Yaskawa INFORM job: LETTERTR.JBI

/JOB
//NAME LETTERTR
//POS
///NPOS 1576,0,0,0,0,0
///TOOL 0
///POSTYPE PULSE
///PULSE
C00000=-2822,58859,-1118,-1041,-34109,-89
C00001=-2663,58398,-451,-1069,-33796,-147
C00002=-2663,58398,-1851,-1069,-33796,-147
C00003=-2764,58391,-1864,-1056,-33791,-106
C00004=-2845,58329,-1958,-1047,-33753,-73
C00005=-2896,58243,-2089,-1041,-33701,-51
C00006=-2915,58143,-2240,-1040,-33641,-43
C00007=-2900,58040,-2395,-1044,-33578,-47
C00008=-2849,57950,-2529,-1052,-33524,-67
C00009=-2767,57884,-2628,-1064,-33484,-99
C00010=-2668,57851,-2677,-1077,-33464,-138
C00011=-2645,57775,-2791,-1081,-33418,-147
C00012=-2722,57704,-2899,-1072,-33375,-115
C00013=-2807,57646,-2987,-1062,-33340,-80
C00014=-2852,57583,-3083,-1057,-33302,-61
C00015=-2760,57536,-3153,-1070,-33273,-98
C00016=-2666,57492,-3219,-1083,-33246,-135
C00017=-2684,57440,-3296,-1081,-33215,-127
C00018=-2776,57397,-3362,-1070,-33190,-90
C00019=-2811,57371,-3402,-1065,-33174,-75
C00020=-2719,57413,-3338,-1077,-33199,-113
C00021=-2626,57455,-3274,-1089,-33224,-150
C00022=-2618,57352,-3429,-1091,-33162,-152
C00023=-2640,57254,-3577,-1090,-33102,-142
C00024=-2673,57160,-3720,-1087,-33045,-128
C00025=-2712,57067,-3860,-1083,-32989,-111
C00026=-2749,56974,-4000,-1080,-32933,-95
C00027=-2729,56988,-3980,-1082,-32941,-103
C00028=-2696,57083,-3836,-1085,-32999,-118
C00029=-2658,57176,-3696,-1089,-33055,-134
C00030=-2620,57268,-3556,-1092,-33111,-150
C00031=-2574,57251,-3581,-1099,-33100,-168
C00032=-2533,57158,-3722,-1106,-33043,-184
C00033=-2487,57065,-3861,-1113,-32987,-201
C00034=-2437,56975,-3997,-1121,-32931,-220
C00035=-2389,56892,-4124,-1129,-32880,-238
C00036=-2428,56983,-3985,-1122,-32936,-224
C00037=-2479,57073,-3849,-1114,-32991,-205
C00038=-2523,57166,-3710,-1107,-33048,-188
C00039=-2565,57259,-3569,-1100,-33105,-172
C00040=-2606,57348,-3435,-1093,-33159,-157
C00041=-2610,57453,-3277,-1091,-33222,-157
C00042=-2508,57437,-3300,-1105,-33213,-197
C00043=-2406,57411,-3339,-1119,-33196,-238
C00044=-2346,57409,-3342,-1127,-33195,-262
C00045=-2448,57433,-3305,-1113,-33210,-221
C00046=-2551,57457,-3270,-1099,-33225,-180
C00047=-2555,57511,-3189,-1097,-33257,-179
C00048=-2468,57564,-3107,-1108,-33290,-215
C00049=-2400,57631,-3005,-1116,-33330,-243
C00050=-2485,57694,-2912,-1104,-33369,-210
C00051=-2569,57757,-2817,-1092,-33407,-177
C00052=-2616,57836,-2698,-1084,-33455,-159
C00053=-2509,57839,-2693,-1098,-33457,-202
C00054=-2413,57872,-2641,-1111,-33477,-241
C00055=-2340,57940,-2537,-1119,-33519,-271
C00056=-2296,58030,-2401,-1124,-33573,-290
C00057=-2288,58130,-2250,-1123,-33634,-294
C00058=-2316,58227,-2102,-1118,-33694,-284
C00059=-2376,58313,-1975,-1109,-33745,-261
C00060=-2460,58376,-1880,-1097,-33784,-228
C00061=-2561,58402,-1842,-1083,-33799,-188
C00062=-2663,58398,-1851,-1069,-33796,-147
C00063=-2663,58398,-451,-1069,-33796,-147
C00064=-2673,58389,-465,-1068,-33790,-142
C00065=-2673,58389,-1865,-1068,-33790,-142
C00066=-2704,58383,-1875,-1064,-33786,-130
C00067=-2673,58381,-1877,-1068,-33785,-143
C00068=-2641,58379,-1880,-1073,-33784,-155
C00069=-2631,58387,-1866,-1074,-33790,-159
C00070=-2599,58391,-1860,-1078,-33792,-172
C00071=-2566,58392,-1859,-1082,-33793,-186
C00072=-2534,58387,-1865,-1087,-33790,-199
C00073=-2502,58380,-1875,-1091,-33786,-211
C00074=-2471,58371,-1889,-1095,-33780,-224
C00075=-2441,58357,-1909,-1099,-33772,-235
C00076=-2416,58336,-1941,-1103,-33759,-245
C00077=-2392,58314,-1973,-1107,-33746,-255
C00078=-2369,58290,-2009,-1110,-33731,-264
C00079=-2346,58266,-2045,-1113,-33717,-272
C00080=-2331,58237,-2088,-1116,-33700,-278
C00081=-2318,58208,-2131,-1118,-33682,-283
C00082=-2306,58179,-2176,-1120,-33664,-288
C00083=-2301,58147,-2224,-1121,-33645,-289
C00084=-2296,58115,-2272,-1122,-33625,-291
C00085=-2294,58082,-2322,-1123,-33605,-291
C00086=-2300,58051,-2369,-1123,-33586,-288
C00087=-2309,58021,-2415,-1122,-33568,-284
C00088=-2321,57993,-2458,-1121,-33551,-279
C00089=-2336,57966,-2499,-1119,-33534,-273
C00090=-2354,57940,-2538,-1117,-33518,-265
C00091=-2372,57914,-2578,-1115,-33503,-258
C00092=-2398,57894,-2607,-1112,-33491,-247
C00093=-2425,57878,-2632,-1109,-33481,-236
C00094=-2453,57864,-2654,-1105,-33472,-224
C00095=-2483,57854,-2669,-1102,-33466,-212
C00096=-2514,57849,-2678,-1098,-33463,-200
C00097=-2548,57848,-2679,-1093,-33462,-186
C00098=-2581,57848,-2680,-1089,-33462,-173
C00099=-2615,57849,-2679,-1084,-33463,-160
C00100=-2646,57857,-2667,-1080,-33468,-147
C00101=-2678,57864,-2657,-1076,-33472,-134
C00102=-2710,57873,-2644,-1071,-33478,-122
C00103=-2739,57885,-2626,-1067,-33485,-110
C00104=-2769,57898,-2606,-1063,-33493,-98
C00105=-2797,57915,-2582,-1059,-33503,-87
C00106=-2821,57936,-2550,-1056,-33516,-78
C00107=-2843,57961,-2512,-1052,-33531,-69
C00108=-2863,57988,-2473,-1049,-33547,-62
C00109=-2877,58017,-2430,-1047,-33564,-56
C00110=-2889,58046,-2385,-1045,-33582,-52
C00111=-2896,58077,-2338,-1044,-33601,-49
C00112=-2900,58110,-2290,-1043,-33621,-48
C00113=-2903,58143,-2240,-1042,-33640,-47
C00114=-2901,58175,-2191,-1041,-33660,-48
C00115=-2893,58206,-2145,-1042,-33679,-52
C00116=-2885,58236,-2099,-1043,-33697,-56
C00117=-2876,58266,-2053,-1043,-33715,-60
C00118=-2860,58293,-2012,-1045,-33732,-66
C00119=-2840,58318,-1974,-1047,-33747,-75
C00120=-2819,58342,-1938,-1050,-33762,-84
C00121=-2793,58361,-1909,-1053,-33773,-94
C00122=-2766,58377,-1884,-1056,-33783,-105
C00123=-2736,58389,-1866,-1060,-33790,-117
C00124=-2705,58393,-1859,-1064,-33793,-130
C00125=-2673,58389,-1865,-1068,-33790,-142
C00126=-2673,58389,-465,-1068,-33790,-142
C00127=-2757,58271,-644,-1059,-33719,-108
C00128=-2757,58271,-2044,-1059,-33719,-108
C00129=-2762,58267,-2051,-1059,-33716,-106
C00130=-2765,58261,-2060,-1058,-33712,-104
C00131=-2768,58254,-2069,-1058,-33709,-103
C00132=-2769,58248,-2080,-1058,-33704,-102
C00133=-2772,58241,-2089,-1058,-33701,-101
C00134=-2773,58234,-2100,-1057,-33696,-101
C00135=-2775,58228,-2110,-1057,-33692,-100
C00136=-2776,58221,-2120,-1057,-33688,-99
C00137=-2778,58214,-2131,-1057,-33684,-98
C00138=-2779,58207,-2141,-1057,-33680,-98
C00139=-2780,58200,-2152,-1057,-33676,-97
C00140=-2781,58193,-2163,-1057,-33671,-97
C00141=-2781,58185,-2174,-1057,-33667,-97
C00142=-2782,58178,-2185,-1057,-33662,-96
C00143=-2782,58171,-2196,-1057,-33658,-96
C00144=-2783,58164,-2206,-1057,-33654,-96
C00145=-2782,58157,-2217,-1057,-33649,-96
C00146=-2781,58150,-2227,-1058,-33645,-97
C00147=-2780,58143,-2238,-1058,-33641,-97
C00148=-2778,58136,-2248,-1058,-33637,-97
C00149=-2776,58129,-2259,-1059,-33633,-98
C00150=-2774,58123,-2268,-1059,-33629,-99
C00151=-2770,58116,-2278,-1060,-33625,-100
C00152=-2767,58110,-2287,-1060,-33621,-102
C00153=-2762,58104,-2296,-1061,-33618,-103
C00154=-2757,58100,-2302,-1062,-33615,-106
C00155=-2750,58097,-2307,-1063,-33613,-108
C00156=-2744,58095,-2310,-1063,-33612,-111
C00157=-2738,58091,-2315,-1064,-33610,-113
C00158=-2731,58090,-2317,-1065,-33609,-116
C00159=-2724,58092,-2314,-1066,-33610,-119
C00160=-2718,58096,-2308,-1067,-33612,-121
C00161=-2713,58100,-2301,-1067,-33615,-123
C00162=-2711,58107,-2291,-1068,-33619,-124
C00163=-2710,58114,-2281,-1068,-33623,-124
C00164=-2708,58120,-2271,-1068,-33627,-125
C00165=-2704,58126,-2262,-1068,-33631,-127
C00166=-2704,58134,-2251,-1068,-33635,-127
C00167=-2704,58141,-2240,-1068,-33640,-127
C00168=-2705,58148,-2229,-1068,-33644,-127
C00169=-2706,58155,-2219,-1067,-33648,-126
C00170=-2707,58162,-2208,-1067,-33653,-126
C00171=-2707,58169,-2198,-1067,-33657,-126
C00172=-2710,58175,-2188,-1067,-33661,-125
C00173=-2710,58183,-2177,-1067,-33665,-126
C00174=-2712,58189,-2167,-1066,-33669,-125
C00175=-2713,58196,-2157,-1066,-33673,-124
C00176=-2716,58202,-2147,-1065,-33677,-123
C00177=-2718,58209,-2137,-1065,-33681,-122
C00178=-2720,58216,-2127,-1065,-33685,-122
C00179=-2722,58222,-2117,-1064,-33689,-121
C00180=-2724,58229,-2107,-1064,-33693,-120
C00181=-2727,58236,-2097,-1064,-33697,-119
C00182=-2733,58239,-2092,-1063,-33699,-117
C00183=-2738,58244,-2084,-1062,-33703,-115
C00184=-2740,58251,-2074,-1062,-33706,-114
C00185=-2743,58257,-2064,-1061,-33710,-113
C00186=-2745,58264,-2054,-1061,-33715,-112
C00187=-2750,58269,-2048,-1060,-33717,-110
C00188=-2757,58271,-2044,-1059,-33719,-108
C00189=-2757,58271,-644,-1059,-33719,-108
C00190=-2516,58232,-699,-1091,-33696,-204
C00191=-2516,58232,-2099,-1091,-33696,-204
C00192=-2518,58225,-2110,-1091,-33691,-203
C00193=-2519,58217,-2121,-1091,-33687,-203
C00194=-2521,58210,-2132,-1091,-33683,-202
C00195=-2522,58203,-2143,-1091,-33678,-201
C00196=-2523,58196,-2154,-1091,-33674,-201
C00197=-2525,58189,-2164,-1091,-33669,-200
C00198=-2526,58181,-2176,-1091,-33665,-199
C00199=-2527,58174,-2187,-1091,-33661,-199
C00200=-2527,58166,-2199,-1091,-33656,-198
C00201=-2527,58158,-2210,-1091,-33651,-198
C00202=-2528,58151,-2222,-1091,-33646,-198
C00203=-2526,58143,-2233,-1091,-33642,-199
C00204=-2525,58136,-2244,-1092,-33637,-199
C00205=-2522,58129,-2254,-1092,-33633,-200
C00206=-2518,58123,-2264,-1093,-33629,-201
C00207=-2516,58116,-2274,-1093,-33625,-202
C00208=-2513,58109,-2285,-1094,-33621,-203
C00209=-2511,58102,-2295,-1094,-33617,-204
C00210=-2507,58096,-2305,-1095,-33613,-206
C00211=-2504,58089,-2314,-1095,-33609,-207
C00212=-2500,58083,-2324,-1096,-33605,-208
C00213=-2495,58077,-2333,-1097,-33601,-210
C00214=-2490,58071,-2342,-1097,-33598,-212
C00215=-2484,58066,-2349,-1098,-33595,-214
C00216=-2478,58063,-2354,-1099,-33593,-217
C00217=-2470,58063,-2354,-1100,-33593,-220
C00218=-2465,58068,-2345,-1101,-33596,-222
C00219=-2462,58074,-2336,-1101,-33600,-224
C00220=-2458,58081,-2327,-1101,-33604,-225
C00221=-2455,58087,-2317,-1102,-33608,-226
C00222=-2453,58094,-2307,-1102,-33612,-228
C00223=-2452,58101,-2295,-1102,-33617,-228
C00224=-2451,58109,-2284,-1102,-33621,-229
C00225=-2450,58116,-2272,-1102,-33626,-229
C00226=-2450,58124,-2261,-1102,-33631,-229
C00227=-2451,58132,-2249,-1102,-33635,-229
C00228=-2451,58140,-2238,-1101,-33640,-229
C00229=-2451,58147,-2226,-1101,-33645,-229
C00230=-2452,58154,-2215,-1101,-33649,-228
C00231=-2453,58162,-2204,-1101,-33653,-228
C00232=-2455,58169,-2193,-1100,-33658,-228
C00233=-2457,58176,-2182,-1100,-33662,-227
C00234=-2458,58183,-2171,-1100,-33666,-226
C00235=-2460,58191,-2160,-1099,-33671,-226
C00236=-2462,58198,-2150,-1099,-33675,-225
C00237=-2464,58205,-2140,-1099,-33679,-224
C00238=-2466,58212,-2129,-1098,-33684,-224
C00239=-2468,58219,-2118,-1098,-33688,-223
C00240=-2470,58226,-2107,-1098,-33692,-222
C00241=-2474,58232,-2098,-1097,-33696,-221
C00242=-2477,58239,-2088,-1096,-33700,-220
C00243=-2479,58246,-2078,-1096,-33704,-219
C00244=-2482,58253,-2067,-1096,-33708,-218
C00245=-2486,58258,-2059,-1095,-33712,-216
C00246=-2494,58260,-2057,-1094,-33713,-213
C00247=-2500,58256,-2063,-1093,-33710,-211
C00248=-2504,58250,-2072,-1093,-33707,-209
C00249=-2508,58244,-2081,-1092,-33703,-207
C00250=-2513,58238,-2090,-1092,-33700,-205
C00251=-2516,58232,-2099,-1091,-33696,-204
C00252=-2516,58232,-699,-1091,-33696,-204
C00253=-2186,58255,-658,-1135,-33711,-337
C00254=-2186,58255,-2058,-1135,-33711,-337
C00255=-2183,58242,-2078,-1135,-33703,-338
C00256=-2179,58229,-2098,-1136,-33695,-339
C00257=-2171,58217,-2115,-1137,-33688,-342
C00258=-2162,58207,-2131,-1138,-33682,-346
C00259=-2150,58199,-2143,-1140,-33677,-350
C00260=-2137,58196,-2148,-1142,-33675,-356
C00261=-2124,58198,-2143,-1144,-33677,-361
C00262=-2112,58204,-2134,-1145,-33680,-366
C00263=-2103,58215,-2118,-1146,-33687,-369
C00264=-2097,58227,-2100,-1147,-33694,-372
C00265=-2098,58239,-2081,-1146,-33701,-372
C00266=-2106,58247,-2069,-1145,-33707,-369
C00267=-2108,58234,-2089,-1145,-33698,-368
C00268=-2111,58221,-2109,-1145,-33690,-366
C00269=-2121,58211,-2124,-1144,-33684,-362
C00270=-2133,58205,-2133,-1142,-33681,-357
C00271=-2147,58206,-2132,-1140,-33681,-352
C00272=-2158,58215,-2118,-1139,-33687,-347
C00273=-2167,58226,-2101,-1138,-33694,-344
C00274=-2173,58239,-2083,-1137,-33701,-342
C00275=-2176,58252,-2063,-1136,-33709,-341
C00276=-2179,58265,-2043,-1135,-33717,-340
C00277=-2181,58279,-2022,-1135,-33726,-339
C00278=-2182,58293,-2001,-1134,-33734,-339
C00279=-2183,58307,-1979,-1134,-33743,-339
C00280=-2181,58321,-1959,-1134,-33751,-340
C00281=-2178,58334,-1939,-1134,-33759,-341
C00282=-2173,58346,-1920,-1135,-33767,-343
C00283=-2168,58359,-1901,-1135,-33774,-345
C00284=-2160,58369,-1885,-1136,-33781,-349
C00285=-2151,58380,-1869,-1137,-33787,-353
C00286=-2138,58385,-1861,-1139,-33791,-358
C00287=-2124,58384,-1862,-1141,-33790,-363
C00288=-2111,58381,-1867,-1142,-33788,-368
C00289=-2104,58370,-1883,-1143,-33782,-371
C00290=-2099,58357,-1902,-1144,-33774,-373
C00291=-2096,58344,-1922,-1145,-33766,-374
C00292=-2093,58330,-1943,-1145,-33757,-375
C00293=-2092,58317,-1964,-1146,-33749,-375
C00294=-2081,58320,-1959,-1147,-33751,-380
C00295=-2082,58333,-1939,-1147,-33759,-379
C00296=-2085,58346,-1919,-1146,-33767,-379
C00297=-2089,58359,-1899,-1146,-33775,-377
C00298=-2093,58372,-1879,-1145,-33783,-376
C00299=-2097,58385,-1860,-1144,-33791,-374
C00300=-2108,58391,-1850,-1143,-33795,-370
C00301=-2122,58395,-1845,-1141,-33797,-364
C00302=-2137,58396,-1844,-1139,-33797,-358
C00303=-2150,58393,-1849,-1137,-33795,-353
C00304=-2161,58385,-1862,-1136,-33790,-348
C00305=-2170,58374,-1878,-1135,-33784,-345
C00306=-2175,58362,-1896,-1134,-33776,-342
C00307=-2182,58351,-1914,-1134,-33769,-340
C00308=-2186,58338,-1933,-1133,-33762,-338
C00309=-2189,58325,-1953,-1133,-33754,-336
C00310=-2191,58311,-1974,-1133,-33745,-335
C00311=-2190,58297,-1995,-1133,-33737,-335
C00312=-2190,58283,-2016,-1134,-33728,-336
C00313=-2188,58269,-2037,-1134,-33720,-336
C00314=-2186,58255,-2058,-1135,-33711,-337
C00315=-2186,58255,-658,-1135,-33711,-337
C00316=-2073,58248,-667,-1150,-33707,-382
C00317=-2073,58248,-2067,-1150,-33707,-382
C00318=-2072,58241,-2077,-1150,-33703,-382
C00319=-2071,58235,-2087,-1150,-33699,-383
C00320=-2069,58229,-2096,-1150,-33695,-383
C00321=-2067,58223,-2105,-1151,-33692,-384
C00322=-2063,58217,-2114,-1151,-33688,-385
C00323=-2059,58212,-2121,-1152,-33685,-387
C00324=-2053,58209,-2126,-1153,-33683,-390
C00325=-2047,58206,-2130,-1154,-33682,-392
C00326=-2041,58203,-2135,-1154,-33680,-394
C00327=-2035,58202,-2137,-1155,-33679,-397
C00328=-2028,58202,-2136,-1156,-33679,-399
C00329=-2021,58202,-2136,-1157,-33679,-402
C00330=-2015,58205,-2131,-1158,-33681,-405
C00331=-2010,58209,-2125,-1158,-33683,-407
C00332=-2006,58214,-2118,-1159,-33687,-409
C00333=-2003,58219,-2109,-1159,-33690,-410
C00334=-2001,58225,-2100,-1159,-33694,-411
C00335=-1999,58231,-2091,-1160,-33697,-412
C00336=-1999,58238,-2080,-1159,-33702,-412
C00337=-1994,58236,-2083,-1160,-33701,-413
C00338=-1993,58230,-2093,-1160,-33697,-414
C00339=-1990,58224,-2101,-1161,-33693,-415
C00340=-1987,58218,-2110,-1161,-33689,-416
C00341=-1985,58212,-2120,-1162,-33686,-417
C00342=-1984,58206,-2129,-1162,-33682,-417
C00343=-1981,58200,-2139,-1162,-33678,-418
C00344=-1976,58196,-2144,-1163,-33676,-420
C00345=-1969,58198,-2142,-1164,-33677,-423
C00346=-1969,58204,-2132,-1164,-33681,-423
C00347=-1973,58209,-2124,-1163,-33684,-422
C00348=-1976,58215,-2115,-1163,-33687,-421
C00349=-1978,58221,-2106,-1162,-33691,-420
C00350=-1980,58227,-2097,-1162,-33695,-419
C00351=-1982,58233,-2088,-1162,-33699,-418
C00352=-1985,58239,-2079,-1161,-33702,-417
C00353=-1987,58245,-2069,-1161,-33706,-417
C00354=-1989,58251,-2060,-1160,-33710,-416
C00355=-1990,58258,-2050,-1160,-33714,-415
C00356=-1992,58264,-2041,-1160,-33718,-415
C00357=-1994,58270,-2032,-1160,-33721,-414
C00358=-1995,58277,-2022,-1159,-33725,-414
C00359=-1998,58283,-2013,-1159,-33729,-413
C00360=-2001,58289,-2004,-1158,-33732,-412
C00361=-2006,58290,-2002,-1158,-33733,-409
C00362=-2012,58292,-2000,-1157,-33734,-407
C00363=-2017,58297,-1992,-1156,-33737,-405
C00364=-2022,58302,-1985,-1155,-33740,-403
C00365=-2029,58303,-1983,-1154,-33741,-401
C00366=-2036,58304,-1982,-1154,-33741,-398
C00367=-2042,58302,-1985,-1153,-33740,-395
C00368=-2047,58298,-1990,-1152,-33738,-393
C00369=-2052,58294,-1997,-1152,-33735,-391
C00370=-2057,58289,-2004,-1151,-33733,-389
C00371=-2061,58284,-2012,-1151,-33729,-387
C00372=-2064,58279,-2020,-1150,-33726,-386
C00373=-2067,58273,-2029,-1150,-33723,-385
C00374=-2069,58267,-2038,-1150,-33719,-384
C00375=-2071,58261,-2047,-1150,-33715,-383
C00376=-2072,58255,-2057,-1150,-33711,-383
C00377=-2073,58248,-2067,-1150,-33707,-382
C00378=-2073,58248,-667,-1150,-33707,-382
C00379=-2064,58248,-666,-1151,-33708,-386
C00380=-2064,58248,-2066,-1151,-33708,-386
C00381=-2063,58252,-2061,-1151,-33710,-386
C00382=-2062,58256,-2055,-1151,-33712,-387
C00383=-2061,58259,-2050,-1151,-33714,-387
C00384=-2060,58263,-2045,-1151,-33716,-388
C00385=-2059,58266,-2039,-1151,-33718,-388
C00386=-2057,58269,-2035,-1151,-33720,-389
C00387=-2056,58273,-2029,-1151,-33722,-389
C00388=-2054,58276,-2024,-1152,-33724,-390
C00389=-2051,58278,-2021,-1152,-33726,-391
C00390=-2050,58281,-2016,-1152,-33728,-392
C00391=-2048,58285,-2011,-1152,-33730,-393
C00392=-2046,58287,-2007,-1152,-33731,-394
C00393=-2042,58289,-2004,-1153,-33733,-395
C00394=-2039,58291,-2001,-1153,-33734,-396
C00395=-2036,58292,-2000,-1154,-33734,-398
C00396=-2032,58293,-1998,-1154,-33735,-399
C00397=-2028,58294,-1997,-1155,-33736,-400
C00398=-2025,58292,-2000,-1155,-33734,-402
C00399=-2022,58289,-2003,-1156,-33733,-403
C00400=-2019,58287,-2007,-1156,-33731,-404
C00401=-2016,58285,-2010,-1156,-33730,-405
C00402=-2013,58282,-2014,-1157,-33729,-407
C00403=-2010,58280,-2017,-1157,-33727,-408
C00404=-2009,58277,-2023,-1158,-33725,-408
C00405=-2008,58273,-2028,-1158,-33723,-409
C00406=-2007,58269,-2033,-1158,-33721,-409
C00407=-2007,58265,-2039,-1158,-33718,-409
C00408=-2006,58262,-2044,-1158,-33716,-409
C00409=-2007,58258,-2050,-1158,-33714,-409
C00410=-2007,58255,-2055,-1158,-33712,-408
C00411=-2007,58251,-2061,-1158,-33709,-409
C00412=-2008,58248,-2067,-1158,-33707,-408
C00413=-2008,58244,-2072,-1158,-33705,-408
C00414=-2008,58240,-2078,-1158,-33702,-408
C00415=-2008,58236,-2084,-1158,-33700,-408
C00416=-2009,58232,-2090,-1158,-33698,-407
C00417=-2010,58229,-2095,-1158,-33696,-407
C00418=-2011,58225,-2101,-1158,-33694,-407
C00419=-2012,58222,-2106,-1158,-33691,-406
C00420=-2015,58219,-2110,-1158,-33690,-405
C00421=-2017,58216,-2115,-1157,-33688,-404
C00422=-2020,58213,-2118,-1157,-33686,-403
C00423=-2023,58211,-2122,-1157,-33685,-402
C00424=-2026,58210,-2124,-1156,-33684,-400
C00425=-2030,58209,-2125,-1156,-33684,-399
C00426=-2034,58210,-2124,-1155,-33684,-397
C00427=-2038,58211,-2123,-1155,-33685,-396
C00428=-2041,58212,-2121,-1154,-33685,-394
C00429=-2045,58213,-2119,-1154,-33686,-393
C00430=-2048,58216,-2116,-1153,-33688,-392
C00431=-2051,58218,-2112,-1153,-33689,-390
C00432=-2054,58220,-2109,-1152,-33690,-389
C00433=-2056,58223,-2104,-1152,-33692,-388
C00434=-2058,58227,-2099,-1152,-33694,-388
C00435=-2060,58230,-2094,-1152,-33696,-387
C00436=-2061,58233,-2089,-1151,-33698,-386
C00437=-2062,58237,-2083,-1151,-33701,-386
C00438=-2062,58241,-2077,-1151,-33703,-386
C00439=-2063,58245,-2072,-1151,-33705,-386
C00440=-2064,58248,-2066,-1151,-33708,-386
C00441=-2064,58248,-666,-1151,-33708,-386
C00442=-1952,58261,-646,-1165,-33715,-431
C00443=-1952,58261,-2046,-1165,-33715,-431
C00444=-1950,58252,-2059,-1166,-33710,-432
C00445=-1948,58243,-2072,-1166,-33705,-432
C00446=-1946,58234,-2086,-1166,-33699,-433
C00447=-1944,58225,-2099,-1167,-33694,-433
C00448=-1943,58216,-2113,-1167,-33688,-434
C00449=-1942,58207,-2127,-1167,-33683,-434
C00450=-1941,58198,-2140,-1168,-33677,-435
C00451=-1936,58190,-2152,-1168,-33672,-436
C00452=-1928,58190,-2152,-1170,-33673,-439
C00453=-1927,58200,-2138,-1169,-33678,-440
C00454=-1929,58208,-2124,-1169,-33684,-439
C00455=-1931,58217,-2111,-1169,-33689,-439
C00456=-1932,58227,-2097,-1169,-33695,-439
C00457=-1932,58236,-2083,-1168,-33700,-438
C00458=-1933,58245,-2069,-1168,-33706,-438
C00459=-1930,58253,-2056,-1168,-33711,-439
C00460=-1927,58262,-2044,-1168,-33716,-441
C00461=-1924,58270,-2032,-1169,-33721,-442
C00462=-1917,58276,-2022,-1170,-33725,-445
C00463=-1908,58279,-2017,-1171,-33727,-449
C00464=-1899,58280,-2015,-1172,-33728,-452
C00465=-1891,58276,-2021,-1173,-33725,-455
C00466=-1884,58270,-2031,-1174,-33721,-458
C00467=-1878,58262,-2042,-1175,-33717,-460
C00468=-1873,58254,-2054,-1176,-33712,-462
C00469=-1870,58246,-2066,-1176,-33707,-464
C00470=-1867,58238,-2079,-1177,-33702,-465
C00471=-1864,58229,-2092,-1177,-33697,-466
C00472=-1862,58220,-2105,-1178,-33691,-466
C00473=-1860,58211,-2119,-1178,-33686,-467
C00474=-1860,58202,-2133,-1178,-33680,-467
C00475=-1856,58194,-2145,-1179,-33675,-468
C00476=-1847,58196,-2142,-1180,-33676,-472
C00477=-1846,58205,-2128,-1180,-33682,-473
C00478=-1848,58214,-2115,-1180,-33687,-472
C00479=-1851,58222,-2102,-1179,-33692,-471
C00480=-1855,58230,-2090,-1179,-33697,-470
C00481=-1857,58239,-2077,-1178,-33703,-469
C00482=-1860,58248,-2064,-1178,-33708,-468
C00483=-1863,58256,-2051,-1177,-33713,-466
C00484=-1867,58264,-2039,-1176,-33718,-465
C00485=-1873,58271,-2028,-1175,-33722,-463
C00486=-1879,58279,-2017,-1175,-33727,-460
C00487=-1886,58285,-2007,-1174,-33731,-458
C00488=-1894,58290,-2000,-1172,-33734,-455
C00489=-1904,58290,-2000,-1171,-33734,-451
C00490=-1912,58288,-2003,-1170,-33733,-447
C00491=-1920,58285,-2008,-1169,-33731,-444
C00492=-1928,58279,-2017,-1168,-33727,-441
C00493=-1933,58272,-2028,-1168,-33723,-439
C00494=-1936,58264,-2040,-1167,-33718,-437
C00495=-1942,58259,-2048,-1167,-33715,-435
C00496=-1945,58268,-2035,-1166,-33720,-434
C00497=-1947,58277,-2022,-1166,-33725,-433
C00498=-1950,58285,-2009,-1165,-33730,-432
C00499=-1955,58292,-1999,-1164,-33734,-430
C00500=-1961,58286,-2007,-1164,-33731,-428
C00501=-1959,58277,-2021,-1164,-33726,-428
C00502=-1956,58269,-2033,-1165,-33721,-429
C00503=-1952,58261,-2046,-1165,-33715,-431
C00504=-1952,58261,-646,-1165,-33715,-431
C00505=-1708,58270,-628,-1197,-33722,-529
C00506=-1708,58270,-2028,-1197,-33722,-529
C00507=-1705,58252,-2054,-1198,-33712,-530
C00508=-1700,58236,-2078,-1199,-33702,-532
C00509=-1693,58220,-2102,-1200,-33692,-534
C00510=-1682,58206,-2123,-1202,-33683,-538
C00511=-1666,58200,-2132,-1204,-33680,-545
C00512=-1651,58208,-2121,-1206,-33684,-551
C00513=-1645,58223,-2098,-1206,-33694,-554
C00514=-1642,58239,-2072,-1206,-33704,-555
C00515=-1645,58257,-2046,-1206,-33714,-554
C00516=-1633,58247,-2061,-1207,-33708,-559
C00517=-1622,58233,-2082,-1209,-33700,-563
C00518=-1612,58218,-2104,-1211,-33691,-567
C00519=-1604,58203,-2127,-1212,-33681,-570
C00520=-1597,58187,-2151,-1213,-33672,-572
C00521=-1595,58170,-2177,-1214,-33661,-573
C00522=-1596,58152,-2204,-1214,-33650,-572
C00523=-1603,58137,-2227,-1213,-33641,-569
C00524=-1611,58123,-2249,-1212,-33632,-566
C00525=-1624,58111,-2268,-1211,-33625,-561
C00526=-1638,58102,-2281,-1209,-33619,-555
C00527=-1655,58105,-2277,-1207,-33621,-548
C00528=-1670,58114,-2263,-1205,-33627,-542
C00529=-1682,58128,-2243,-1203,-33635,-537
C00530=-1694,58142,-2221,-1201,-33644,-533
C00531=-1703,58157,-2199,-1200,-33653,-530
C00532=-1710,58169,-2180,-1199,-33660,-527
C00533=-1705,58153,-2205,-1200,-33650,-529
C00534=-1697,58138,-2228,-1201,-33641,-532
C00535=-1687,58123,-2250,-1203,-33632,-536
C00536=-1675,58110,-2270,-1204,-33624,-540
C00537=-1661,58099,-2286,-1206,-33617,-546
C00538=-1644,58094,-2293,-1209,-33614,-552
C00539=-1627,58097,-2289,-1211,-33616,-559
C00540=-1612,58106,-2275,-1213,-33622,-565
C00541=-1601,58119,-2255,-1214,-33630,-570
C00542=-1592,58133,-2233,-1215,-33639,-574
C00543=-1587,58149,-2209,-1215,-33648,-576
C00544=-1584,58166,-2183,-1215,-33659,-578
C00545=-1586,58183,-2157,-1215,-33669,-577
C00546=-1591,58199,-2133,-1214,-33679,-575
C00547=-1598,58215,-2109,-1213,-33689,-572
C00548=-1607,58230,-2086,-1211,-33698,-569
C00549=-1617,58244,-2065,-1210,-33707,-565
C00550=-1628,58258,-2044,-1208,-33715,-561
C00551=-1640,58272,-2023,-1206,-33724,-556
C00552=-1648,58287,-2000,-1205,-33733,-553
C00553=-1658,58282,-2009,-1204,-33730,-549
C00554=-1654,58265,-2034,-1204,-33720,-551
C00555=-1652,58248,-2060,-1205,-33709,-551
C00556=-1651,58231,-2086,-1205,-33698,-551
C00557=-1656,58215,-2110,-1205,-33689,-549
C00558=-1671,58211,-2116,-1203,-33686,-543
C00559=-1683,58222,-2099,-1201,-33693,-538
C00560=-1690,58238,-2075,-1200,-33703,-536
C00561=-1694,58255,-2050,-1199,-33713,-534
C00562=-1697,58272,-2024,-1199,-33723,-533
C00563=-1697,58290,-1997,-1198,-33735,-534
C00564=-1705,58303,-1978,-1197,-33742,-530
C00565=-1709,58287,-2001,-1197,-33733,-529
C00566=-1708,58270,-2028,-1197,-33722,-529
C00567=-1708,58270,-628,-1197,-33722,-529
C00568=-1590,58245,-662,-1213,-33708,-576
C00569=-1590,58245,-2062,-1213,-33708,-576
C00570=-1592,58236,-2076,-1213,-33702,-575
C00571=-1593,58227,-2090,-1213,-33696,-575
C00572=-1592,58218,-2104,-1213,-33691,-575
C00573=-1588,58209,-2118,-1214,-33685,-576
C00574=-1586,58200,-2131,-1215,-33680,-577
C00575=-1579,58193,-2142,-1215,-33675,-580
C00576=-1574,58185,-2155,-1216,-33670,-582
C00577=-1568,58178,-2165,-1217,-33666,-584
C00578=-1560,58172,-2174,-1218,-33663,-587
C00579=-1551,58168,-2179,-1220,-33661,-591
C00580=-1542,58166,-2182,-1221,-33659,-594
C00581=-1532,58166,-2181,-1222,-33659,-598
C00582=-1523,58169,-2176,-1223,-33661,-602
C00583=-1516,58174,-2169,-1224,-33664,-605
C00584=-1511,58182,-2157,-1225,-33669,-607
C00585=-1509,58191,-2144,-1225,-33675,-608
C00586=-1508,58200,-2129,-1225,-33680,-608
C00587=-1509,58210,-2115,-1224,-33686,-608
C00588=-1511,58219,-2101,-1224,-33692,-608
C00589=-1513,58228,-2087,-1224,-33697,-607
C00590=-1517,58237,-2074,-1223,-33703,-605
C00591=-1520,58245,-2061,-1222,-33708,-604
C00592=-1526,58253,-2049,-1221,-33713,-602
C00593=-1531,58261,-2037,-1221,-33718,-600
C00594=-1538,58268,-2026,-1220,-33722,-597
C00595=-1544,58276,-2015,-1219,-33727,-595
C00596=-1552,58281,-2007,-1218,-33730,-592
C00597=-1550,58272,-2021,-1218,-33724,-592
C00598=-1543,58265,-2032,-1219,-33720,-595
C00599=-1537,58257,-2043,-1220,-33715,-597
C00600=-1532,58249,-2056,-1221,-33710,-599
C00601=-1528,58241,-2068,-1221,-33705,-601
C00602=-1524,58232,-2081,-1222,-33700,-602
C00603=-1521,58224,-2094,-1223,-33695,-604
C00604=-1519,58215,-2108,-1223,-33689,-604
C00605=-1517,58205,-2122,-1223,-33683,-605
C00606=-1518,58196,-2136,-1223,-33678,-604
C00607=-1520,58187,-2150,-1223,-33672,-603
C00608=-1526,58180,-2161,-1223,-33668,-601
C00609=-1534,58177,-2166,-1222,-33666,-597
C00610=-1544,58177,-2165,-1220,-33666,-594
C00611=-1553,58180,-2162,-1219,-33667,-590
C00612=-1561,58185,-2153,-1218,-33671,-587
C00613=-1567,58192,-2143,-1217,-33675,-584
C00614=-1572,58200,-2131,-1216,-33680,-582
C00615=-1577,58208,-2118,-1215,-33685,-581
C00616=-1580,58217,-2105,-1215,-33690,-580
C00617=-1582,58226,-2091,-1215,-33696,-579
C00618=-1581,58236,-2077,-1215,-33702,-580
C00619=-1579,58245,-2063,-1215,-33707,-581
C00620=-1574,58252,-2051,-1215,-33712,-583
C00621=-1567,58259,-2042,-1216,-33716,-586
C00622=-1558,58260,-2040,-1217,-33717,-589
C00623=-1552,58259,-2042,-1218,-33716,-592
C00624=-1556,58267,-2029,-1217,-33721,-590
C00625=-1565,58270,-2025,-1216,-33723,-587
C00626=-1573,58267,-2029,-1215,-33721,-583
C00627=-1581,58261,-2038,-1214,-33718,-580
C00628=-1586,58254,-2050,-1214,-33713,-578
C00629=-1590,58245,-2062,-1213,-33708,-576
C00630=-1590,58245,-662,-1213,-33708,-576
C00631=-1499,58245,-662,-1225,-33708,-613
C00632=-1499,58245,-2062,-1225,-33708,-613
C00633=-1497,58235,-2076,-1226,-33702,-613
C00634=-1495,58226,-2090,-1226,-33696,-614
C00635=-1493,58217,-2104,-1226,-33691,-615
C00636=-1490,58208,-2118,-1227,-33685,-616
C00637=-1487,58199,-2131,-1228,-33680,-617
C00638=-1481,58191,-2143,-1228,-33675,-619
C00639=-1476,58183,-2155,-1229,-33670,-621
C00640=-1468,58176,-2165,-1230,-33666,-624
C00641=-1460,58171,-2174,-1232,-33662,-627
C00642=-1452,58166,-2181,-1233,-33659,-630
C00643=-1444,58161,-2187,-1234,-33657,-634
C00644=-1434,58160,-2189,-1235,-33656,-637
C00645=-1424,58160,-2190,-1236,-33656,-641
C00646=-1415,58162,-2186,-1238,-33657,-645
C00647=-1408,58169,-2176,-1238,-33661,-648
C00648=-1404,58176,-2164,-1239,-33666,-650
C00649=-1401,58185,-2151,-1239,-33671,-651
C00650=-1400,58195,-2136,-1239,-33677,-652
C00651=-1399,58204,-2121,-1239,-33683,-652
C00652=-1399,58214,-2106,-1239,-33689,-653
C00653=-1399,58224,-2092,-1239,-33695,-652
C00654=-1402,58233,-2078,-1238,-33701,-651
C00655=-1404,58242,-2064,-1238,-33707,-651
C00656=-1407,58251,-2050,-1237,-33712,-650
C00657=-1410,58260,-2037,-1237,-33718,-649
C00658=-1413,58269,-2023,-1236,-33723,-648
C00659=-1417,58277,-2010,-1235,-33728,-646
C00660=-1422,58285,-1999,-1235,-33733,-644
C00661=-1429,58291,-1990,-1234,-33737,-641
C00662=-1429,58282,-2004,-1234,-33731,-641
C00663=-1425,58273,-2017,-1234,-33726,-643
C00664=-1421,58265,-2030,-1235,-33720,-644
C00665=-1418,58256,-2043,-1236,-33715,-645
C00666=-1416,58247,-2057,-1236,-33709,-646
C00667=-1413,58238,-2071,-1237,-33704,-647
C00668=-1411,58229,-2085,-1237,-33698,-648
C00669=-1409,58219,-2099,-1237,-33692,-649
C00670=-1409,58210,-2113,-1238,-33687,-648
C00671=-1409,58200,-2128,-1238,-33681,-648
C00672=-1411,58191,-2142,-1238,-33675,-647
C00673=-1413,58182,-2156,-1238,-33669,-646
C00674=-1417,58174,-2168,-1237,-33664,-644
C00675=-1426,58169,-2175,-1236,-33662,-641
C00676=-1435,58169,-2175,-1235,-33661,-637
C00677=-1444,58173,-2170,-1234,-33664,-634
C00678=-1452,58178,-2162,-1232,-33667,-630
C00679=-1460,58184,-2154,-1231,-33670,-627
C00680=-1468,58190,-2144,-1230,-33674,-624
C00681=-1474,58198,-2132,-1229,-33679,-622
C00682=-1478,58207,-2119,-1229,-33684,-620
C00683=-1482,58215,-2106,-1228,-33690,-619
C00684=-1484,58224,-2092,-1227,-33695,-618
C00685=-1486,58234,-2078,-1227,-33701,-618
C00686=-1488,58243,-2064,-1227,-33707,-617
C00687=-1490,58252,-2050,-1226,-33713,-617
C00688=-1489,58262,-2034,-1226,-33719,-617
C00689=-1495,58269,-2025,-1225,-33722,-614
C00690=-1502,58263,-2034,-1224,-33719,-612
C00691=-1500,58254,-2047,-1225,-33714,-612
C00692=-1499,58245,-2062,-1225,-33708,-613
C00693=-1499,58245,-662,-1225,-33708,-613
C00694=-1517,58080,-913,-1226,-33606,-603
C00695=-1517,58080,-2313,-1226,-33606,-603
C00696=-1518,58057,-2347,-1226,-33592,-603
C00697=-1512,58035,-2380,-1227,-33579,-604
C00698=-1507,58014,-2413,-1228,-33565,-606
C00699=-1510,57996,-2440,-1228,-33554,-605
C00700=-1534,57998,-2437,-1225,-33556,-595
C00701=-1541,57990,-2449,-1224,-33551,-592
C00702=-1518,57987,-2454,-1227,-33549,-602
C00703=-1501,57976,-2470,-1230,-33542,-608
C00704=-1497,57954,-2503,-1230,-33529,-609
C00705=-1494,57932,-2538,-1231,-33515,-610
C00706=-1495,57909,-2573,-1232,-33501,-610
C00707=-1483,57902,-2582,-1233,-33497,-614
C00708=-1484,57925,-2548,-1233,-33511,-614
C00709=-1486,57948,-2513,-1232,-33525,-614
C00710=-1490,57970,-2479,-1231,-33538,-612
C00711=-1487,57988,-2452,-1231,-33549,-614
C00712=-1464,57990,-2448,-1234,-33551,-623
C00713=-1443,57999,-2435,-1237,-33556,-632
C00714=-1431,57989,-2450,-1239,-33550,-636
C00715=-1424,57967,-2482,-1240,-33537,-639
C00716=-1418,57946,-2515,-1241,-33524,-641
C00717=-1414,57924,-2549,-1242,-33510,-642
C00718=-1413,57901,-2584,-1243,-33496,-642
C00719=-1401,57891,-2598,-1244,-33490,-647
C00720=-1401,57914,-2563,-1244,-33504,-647
C00721=-1403,57937,-2528,-1243,-33518,-647
C00722=-1401,57960,-2493,-1243,-33533,-648
C00723=-1392,57980,-2463,-1244,-33545,-652
C00724=-1375,57994,-2442,-1246,-33553,-659
C00725=-1355,57983,-2458,-1249,-33547,-667
C00726=-1342,57964,-2486,-1251,-33535,-672
C00727=-1334,57943,-2518,-1252,-33522,-675
C00728=-1329,57921,-2551,-1253,-33509,-676
C00729=-1325,57899,-2585,-1254,-33495,-677
C00730=-1320,57878,-2618,-1255,-33482,-679
C00731=-1313,57893,-2594,-1256,-33491,-682
C00732=-1318,57915,-2561,-1255,-33505,-681
C00733=-1322,57937,-2527,-1254,-33518,-679
C00734=-1329,57958,-2495,-1253,-33531,-677
C00735=-1338,57978,-2464,-1251,-33544,-673
C00736=-1355,57995,-2439,-1249,-33554,-667
C00737=-1376,58003,-2428,-1246,-33559,-659
C00738=-1394,57990,-2448,-1243,-33551,-651
C00739=-1405,57971,-2477,-1242,-33539,-647
C00740=-1414,57967,-2483,-1241,-33537,-643
C00741=-1420,57988,-2450,-1240,-33550,-641
C00742=-1426,58010,-2417,-1239,-33563,-639
C00743=-1434,58031,-2386,-1237,-33576,-636
C00744=-1442,58052,-2354,-1236,-33589,-633
C00745=-1450,58073,-2323,-1235,-33602,-630
C00746=-1454,58056,-2347,-1234,-33592,-628
C00747=-1447,58035,-2379,-1236,-33579,-631
C00748=-1439,58014,-2411,-1237,-33566,-634
C00749=-1449,58002,-2430,-1236,-33558,-629
C00750=-1471,57997,-2437,-1233,-33555,-620
C00751=-1495,57999,-2436,-1230,-33556,-611
C00752=-1499,58021,-2402,-1229,-33570,-610
C00753=-1504,58043,-2369,-1228,-33583,-608
C00754=-1506,58065,-2334,-1227,-33597,-607
C00755=-1517,58080,-2313,-1226,-33606,-603
C00756=-1517,58080,-913,-1226,-33606,-603
C00757=-1656,58032,-988,-1208,-33576,-547
C00758=-1656,58032,-2388,-1208,-33576,-547
C00759=-1666,58040,-2376,-1207,-33581,-543
C00760=-1678,58045,-2368,-1205,-33584,-538
C00761=-1692,58046,-2367,-1203,-33585,-532
C00762=-1704,58042,-2373,-1202,-33582,-527
C00763=-1714,58035,-2385,-1200,-33578,-523
C00764=-1723,58025,-2400,-1199,-33572,-520
C00765=-1729,58014,-2417,-1199,-33565,-517
C00766=-1734,58002,-2434,-1198,-33558,-515
C00767=-1738,57990,-2452,-1198,-33550,-513
C00768=-1741,57978,-2471,-1198,-33543,-512
C00769=-1741,57965,-2491,-1198,-33535,-512
C00770=-1739,57952,-2511,-1199,-33527,-512
C00771=-1736,57939,-2530,-1199,-33519,-513
C00772=-1729,57928,-2546,-1200,-33512,-516
C00773=-1719,57919,-2561,-1202,-33507,-520
C00774=-1706,57914,-2567,-1203,-33504,-525
C00775=-1694,57911,-2573,-1205,-33502,-530
C00776=-1680,57908,-2576,-1207,-33500,-535
C00777=-1667,57909,-2574,-1209,-33501,-540
C00778=-1654,57911,-2571,-1210,-33502,-546
C00779=-1642,57916,-2564,-1212,-33505,-550
C00780=-1632,57924,-2551,-1213,-33510,-555
C00781=-1624,57934,-2536,-1214,-33516,-558
C00782=-1617,57945,-2519,-1215,-33523,-561
C00783=-1616,57953,-2508,-1215,-33527,-562
C00784=-1625,57943,-2522,-1214,-33522,-558
C00785=-1634,57934,-2536,-1213,-33516,-554
C00786=-1644,57926,-2549,-1212,-33511,-550
C00787=-1656,57921,-2556,-1210,-33508,-545
C00788=-1669,57919,-2560,-1208,-33507,-540
C00789=-1682,57918,-2561,-1207,-33506,-535
C00790=-1695,57922,-2556,-1205,-33508,-529
C00791=-1707,57926,-2550,-1203,-33511,-525
C00792=-1718,57933,-2539,-1202,-33515,-520
C00793=-1727,57944,-2522,-1200,-33522,-517
C00794=-1731,57956,-2504,-1200,-33530,-516
C00795=-1731,57970,-2483,-1199,-33538,-516
C00796=-1730,57982,-2465,-1199,-33545,-516
C00797=-1726,57994,-2446,-1199,-33553,-518
C00798=-1722,58006,-2428,-1200,-33560,-520
C00799=-1716,58017,-2411,-1200,-33567,-522
C00800=-1707,58027,-2396,-1201,-33573,-526
C00801=-1697,58035,-2384,-1203,-33578,-530
C00802=-1684,58037,-2380,-1204,-33579,-535
C00803=-1672,58034,-2385,-1206,-33577,-540
C00804=-1662,58025,-2398,-1207,-33572,-544
C00805=-1658,58013,-2417,-1208,-33564,-545
C00806=-1665,58002,-2433,-1207,-33558,-542
C00807=-1678,57999,-2439,-1206,-33556,-537
C00808=-1691,57998,-2440,-1204,-33555,-532
C00809=-1704,57997,-2441,-1202,-33555,-527
C00810=-1716,57997,-2442,-1201,-33554,-522
C00811=-1708,57989,-2454,-1202,-33549,-525
C00812=-1695,57989,-2454,-1204,-33550,-531
C00813=-1681,57989,-2454,-1206,-33550,-536
C00814=-1669,57993,-2447,-1207,-33552,-541
C00815=-1657,57997,-2440,-1209,-33555,-546
C00816=-1650,58007,-2425,-1209,-33561,-549
C00817=-1650,58020,-2405,-1209,-33569,-549
C00818=-1656,58032,-2388,-1208,-33576,-547
C00819=-1656,58032,-988,-1208,-33576,-547
C00820=-1764,58027,-997,-1194,-33573,-503
C00821=-1764,58027,-2397,-1194,-33573,-503
C00822=-1767,58034,-2386,-1193,-33577,-502
C00823=-1773,58041,-2376,-1193,-33582,-500
C00824=-1779,58047,-2367,-1192,-33585,-497
C00825=-1787,58049,-2363,-1191,-33587,-494
C00826=-1796,58051,-2362,-1189,-33587,-491
C00827=-1803,58048,-2365,-1188,-33586,-488
C00828=-1812,58047,-2367,-1187,-33585,-484
C00829=-1819,58044,-2372,-1186,-33583,-481
C00830=-1826,58039,-2380,-1186,-33580,-479
C00831=-1830,58033,-2390,-1185,-33576,-477
C00832=-1834,58026,-2400,-1185,-33572,-475
C00833=-1838,58018,-2411,-1184,-33567,-473
C00834=-1840,58011,-2423,-1184,-33563,-472
C00835=-1841,58002,-2436,-1184,-33558,-472
C00836=-1843,57994,-2448,-1184,-33553,-471
C00837=-1843,57986,-2461,-1184,-33547,-471
C00838=-1842,57977,-2474,-1184,-33542,-471
C00839=-1842,57969,-2486,-1185,-33537,-471
C00840=-1839,57961,-2498,-1185,-33532,-472
C00841=-1835,57954,-2509,-1186,-33528,-474
C00842=-1830,57947,-2520,-1187,-33523,-475
C00843=-1824,57942,-2528,-1188,-33520,-478
C00844=-1816,57938,-2533,-1189,-33518,-481
C00845=-1808,57937,-2535,-1190,-33517,-484
C00846=-1799,57936,-2536,-1191,-33517,-488
C00847=-1790,57936,-2536,-1192,-33517,-491
C00848=-1782,57937,-2533,-1193,-33518,-495
C00849=-1774,57940,-2530,-1194,-33519,-498
C00850=-1767,57944,-2524,-1195,-33522,-501
C00851=-1760,57947,-2518,-1196,-33524,-504
C00852=-1753,57952,-2511,-1197,-33527,-507
C00853=-1747,57957,-2503,-1197,-33530,-509
C00854=-1754,57956,-2504,-1196,-33530,-506
C00855=-1761,57953,-2510,-1196,-33527,-503
C00856=-1769,57950,-2514,-1195,-33526,-500
C00857=-1776,57947,-2519,-1194,-33524,-497
C00858=-1784,57945,-2522,-1193,-33522,-494
C00859=-1793,57944,-2523,-1192,-33522,-491
C00860=-1802,57945,-2522,-1190,-33522,-487
C00861=-1810,57946,-2520,-1189,-33523,-484
C00862=-1818,57949,-2516,-1188,-33525,-481
C00863=-1824,57955,-2508,-1187,-33528,-478
C00864=-1828,57962,-2497,-1187,-33533,-477
C00865=-1831,57970,-2485,-1186,-33538,-475
C00866=-1833,57978,-2473,-1186,-33542,-475
C00867=-1832,57986,-2460,-1186,-33547,-475
C00868=-1832,57995,-2447,-1186,-33553,-475
C00869=-1831,58003,-2435,-1186,-33558,-476
C00870=-1829,58011,-2423,-1186,-33563,-477
C00871=-1826,58018,-2411,-1186,-33567,-478
C00872=-1822,58025,-2401,-1186,-33572,-480
C00873=-1817,58032,-2391,-1187,-33576,-482
C00874=-1810,58036,-2384,-1188,-33578,-485
C00875=-1802,58038,-2380,-1189,-33580,-488
C00876=-1794,58040,-2378,-1190,-33581,-491
C00877=-1786,58039,-2379,-1191,-33580,-495
C00878=-1778,58036,-2384,-1192,-33578,-498
C00879=-1773,58029,-2394,-1193,-33574,-499
C00880=-1766,58024,-2402,-1194,-33571,-502
C00881=-1764,58027,-2397,-1194,-33573,-503
C00882=-1764,58027,-997,-1194,-33573,-503
C00883=-1889,58021,-1009,-1178,-33569,-453
C00884=-1889,58021,-2409,-1178,-33569,-453
C00885=-1892,58027,-2398,-1177,-33573,-452
C00886=-1895,58034,-2388,-1177,-33577,-451
C00887=-1899,58040,-2379,-1176,-33581,-449
C00888=-1905,58046,-2371,-1175,-33584,-447
C00889=-1910,58052,-2362,-1174,-33588,-445
C00890=-1916,58056,-2356,-1173,-33590,-442
C00891=-1924,58056,-2355,-1172,-33590,-439
C00892=-1932,58054,-2359,-1171,-33589,-436
C00893=-1938,58051,-2364,-1171,-33587,-434
C00894=-1944,58047,-2370,-1170,-33585,-431
C00895=-1950,58041,-2378,-1169,-33581,-429
C00896=-1956,58037,-2385,-1168,-33579,-426
C00897=-1961,58031,-2394,-1168,-33575,-424
C00898=-1964,58025,-2403,-1167,-33571,-423
C00899=-1968,58019,-2413,-1167,-33567,-421
C00900=-1971,58012,-2423,-1167,-33563,-420
C00901=-1974,58006,-2433,-1167,-33559,-419
C00902=-1976,57999,-2444,-1166,-33555,-418
C00903=-1977,57991,-2456,-1166,-33550,-417
C00904=-1978,57984,-2466,-1166,-33546,-417
C00905=-1977,57976,-2478,-1167,-33541,-417
C00906=-1975,57969,-2489,-1167,-33537,-418
C00907=-1973,57962,-2499,-1167,-33532,-419
C00908=-1969,57955,-2509,-1168,-33528,-420
C00909=-1965,57949,-2519,-1169,-33524,-421
C00910=-1960,57942,-2529,-1169,-33521,-423
C00911=-1954,57937,-2537,-1170,-33517,-426
C00912=-1948,57934,-2541,-1171,-33515,-428
C00913=-1940,57932,-2545,-1172,-33514,-431
C00914=-1933,57932,-2544,-1173,-33514,-434
C00915=-1926,57933,-2543,-1174,-33515,-437
C00916=-1920,57936,-2537,-1175,-33517,-439
C00917=-1914,57941,-2531,-1176,-33520,-442
C00918=-1909,57946,-2522,-1176,-33523,-444
C00919=-1903,57952,-2514,-1177,-33526,-446
C00920=-1900,57958,-2503,-1177,-33530,-448
C00921=-1897,57965,-2493,-1177,-33534,-449
C00922=-1896,57972,-2482,-1177,-33539,-450
C00923=-1895,57980,-2470,-1177,-33544,-450
C00924=-1891,57984,-2465,-1178,-33546,-452
C00925=-1889,57976,-2476,-1178,-33542,-452
C00926=-1887,57969,-2487,-1179,-33537,-453
C00927=-1885,57962,-2498,-1179,-33533,-454
C00928=-1883,57955,-2508,-1179,-33528,-455
C00929=-1881,57948,-2519,-1180,-33524,-455
C00930=-1879,57940,-2530,-1180,-33519,-456
C00931=-1873,57936,-2537,-1181,-33517,-458
C00932=-1865,57937,-2536,-1182,-33517,-461
C00933=-1863,57943,-2526,-1182,-33521,-462
C00934=-1868,57949,-2517,-1182,-33525,-460
C00935=-1871,57955,-2507,-1181,-33529,-459
C00936=-1873,57963,-2496,-1181,-33533,-458
C00937=-1875,57970,-2485,-1180,-33538,-458
C00938=-1878,57977,-2475,-1180,-33542,-457
C00939=-1879,57984,-2464,-1179,-33546,-456
C00940=-1881,57992,-2453,-1179,-33551,-456
C00941=-1883,57999,-2441,-1179,-33555,-455
C00942=-1884,58006,-2430,-1178,-33560,-455
C00943=-1887,58013,-2420,-1178,-33564,-454
C00944=-1889,58021,-2409,-1178,-33569,-453
C00945=-1889,58021,-1009,-1178,-33569,-453
C00946=-1904,58018,-1013,-1176,-33567,-447
C00947=-1904,58018,-2413,-1176,-33567,-447
C00948=-1903,58014,-2419,-1176,-33564,-447
C00949=-1903,58009,-2427,-1176,-33561,-447
C00950=-1902,58005,-2433,-1176,-33559,-447
C00951=-1902,58000,-2440,-1176,-33556,-447
C00952=-1902,57995,-2447,-1176,-33553,-447
C00953=-1901,57991,-2454,-1176,-33550,-447
C00954=-1902,57986,-2462,-1176,-33547,-447
C00955=-1903,57982,-2468,-1176,-33545,-447
C00956=-1903,57977,-2475,-1176,-33542,-447
C00957=-1904,57973,-2482,-1176,-33539,-446
C00958=-1905,57968,-2488,-1176,-33536,-446
C00959=-1906,57964,-2495,-1176,-33534,-445
C00960=-1908,57960,-2501,-1176,-33531,-445
C00961=-1910,57956,-2506,-1176,-33529,-444
C00962=-1913,57953,-2512,-1175,-33527,-442
C00963=-1916,57950,-2517,-1175,-33525,-441
C00964=-1920,57947,-2521,-1175,-33523,-440
C00965=-1923,57944,-2526,-1174,-33521,-438
C00966=-1927,57942,-2529,-1174,-33520,-437
C00967=-1931,57941,-2530,-1173,-33520,-435
C00968=-1936,57940,-2531,-1173,-33519,-433
C00969=-1940,57940,-2531,-1172,-33519,-431
C00970=-1944,57942,-2529,-1172,-33520,-430
C00971=-1948,57944,-2525,-1171,-33522,-428
C00972=-1952,57947,-2521,-1170,-33524,-427
C00973=-1955,57951,-2515,-1170,-33526,-426
C00974=-1957,57955,-2510,-1170,-33528,-425
C00975=-1959,57959,-2504,-1169,-33531,-424
C00976=-1961,57963,-2497,-1169,-33533,-423
C00977=-1964,57967,-2492,-1169,-33535,-422
C00978=-1965,57971,-2485,-1168,-33538,-422
C00979=-1966,57976,-2478,-1168,-33541,-422
C00980=-1967,57980,-2472,-1168,-33544,-421
C00981=-1966,57985,-2464,-1168,-33546,-421
C00982=-1966,57989,-2457,-1168,-33549,-421
C00983=-1965,57994,-2451,-1168,-33552,-422
C00984=-1965,57998,-2444,-1168,-33555,-422
C00985=-1964,58003,-2437,-1168,-33557,-423
C00986=-1962,58007,-2431,-1168,-33560,-423
C00987=-1961,58011,-2425,-1168,-33562,-424
C00988=-1958,58014,-2419,-1168,-33565,-425
C00989=-1955,58018,-2414,-1169,-33567,-426
C00990=-1953,58022,-2408,-1169,-33569,-427
C00991=-1951,58025,-2403,-1169,-33571,-428
C00992=-1948,58029,-2397,-1170,-33573,-429
C00993=-1944,58032,-2393,-1170,-33575,-431
C00994=-1940,58034,-2389,-1171,-33577,-432
C00995=-1937,58038,-2384,-1171,-33579,-434
C00996=-1934,58041,-2379,-1171,-33581,-435
C00997=-1930,58043,-2376,-1172,-33582,-437
C00998=-1926,58044,-2373,-1172,-33583,-439
C00999=-1921,58045,-2372,-1173,-33584,-440
C01000=-1916,58044,-2373,-1174,-33583,-442
C01001=-1912,58043,-2376,-1174,-33582,-444
C01002=-1908,58040,-2379,-1175,-33581,-445
C01003=-1907,58036,-2386,-1175,-33578,-446
C01004=-1906,58031,-2393,-1175,-33575,-446
C01005=-1906,58027,-2399,-1175,-33572,-446
C01006=-1905,58023,-2406,-1175,-33570,-447
C01007=-1904,58018,-2413,-1176,-33567,-447
C01008=-1904,58018,-1013,-1176,-33567,-447
C01009=-1981,58055,-958,-1165,-33589,-416
C01010=-1981,58055,-2358,-1165,-33589,-416
C01011=-1996,58062,-2348,-1163,-33594,-411
C01012=-2011,58056,-2356,-1161,-33590,-405
C01013=-2021,58044,-2376,-1160,-33582,-400
C01014=-2028,58029,-2398,-1159,-33574,-397
C01015=-2034,58014,-2420,-1159,-33564,-395
C01016=-2040,58015,-2419,-1158,-33565,-392
C01017=-2044,58031,-2396,-1157,-33575,-391
C01018=-2046,58048,-2370,-1156,-33585,-390
C01019=-2058,58047,-2371,-1155,-33584,-385
C01020=-2071,58043,-2378,-1153,-33582,-380
C01021=-2087,58038,-2386,-1151,-33579,-374
C01022=-2104,58036,-2389,-1149,-33578,-367
C01023=-2120,58032,-2394,-1147,-33575,-360
C01024=-2124,58048,-2371,-1146,-33585,-359
C01025=-2128,58064,-2347,-1145,-33594,-357
C01026=-2133,58079,-2324,-1144,-33604,-356
C01027=-2138,58095,-2300,-1143,-33614,-354
C01028=-2147,58108,-2281,-1142,-33621,-351
C01029=-2149,58093,-2304,-1142,-33612,-350
C01030=-2145,58077,-2328,-1143,-33602,-351
C01031=-2138,58062,-2350,-1144,-33593,-353
C01032=-2135,58045,-2375,-1145,-33583,-354
C01033=-2134,58030,-2399,-1145,-33574,-355
C01034=-2151,58028,-2402,-1143,-33572,-348
C01035=-2168,58027,-2403,-1141,-33572,-341
C01036=-2184,58024,-2408,-1138,-33570,-334
C01037=-2190,58014,-2424,-1138,-33564,-332
C01038=-2174,58016,-2420,-1140,-33565,-339
C01039=-2157,58017,-2418,-1142,-33566,-345
C01040=-2140,58019,-2415,-1144,-33567,-352
C01041=-2130,58012,-2425,-1146,-33563,-356
C01042=-2128,57996,-2450,-1146,-33553,-356
C01043=-2128,57978,-2476,-1147,-33542,-356
C01044=-2129,57961,-2502,-1147,-33532,-356
C01045=-2126,57945,-2527,-1147,-33522,-357
C01046=-2115,57951,-2518,-1149,-33526,-361
C01047=-2118,57967,-2493,-1148,-33536,-360
C01048=-2118,57985,-2466,-1148,-33546,-361
C01049=-2118,58002,-2440,-1148,-33557,-361
C01050=-2120,58019,-2415,-1147,-33567,-360
C01051=-2107,58025,-2405,-1149,-33571,-365
C01052=-2091,58029,-2399,-1151,-33573,-372
C01053=-2075,58032,-2395,-1153,-33575,-378
C01054=-2060,58037,-2386,-1155,-33578,-385
C01055=-2054,58023,-2408,-1156,-33570,-387
C01056=-2050,58007,-2432,-1157,-33560,-388
C01057=-2047,57991,-2457,-1157,-33550,-389
C01058=-2045,57974,-2482,-1158,-33540,-389
C01059=-2046,57957,-2507,-1158,-33529,-389
C01060=-2045,57940,-2533,-1158,-33519,-389
C01061=-2033,57940,-2533,-1160,-33519,-394
C01062=-2031,57957,-2507,-1160,-33529,-395
C01063=-2032,57974,-2482,-1159,-33540,-395
C01064=-2029,57991,-2456,-1159,-33550,-396
C01065=-2026,58006,-2433,-1160,-33560,-398
C01066=-2021,58022,-2409,-1160,-33569,-400
C01067=-2016,58037,-2387,-1161,-33578,-402
C01068=-2006,58050,-2367,-1162,-33586,-406
C01069=-1991,58053,-2361,-1164,-33588,-413
C01070=-1981,58055,-2358,-1165,-33589,-416
C01071=-1981,58055,-958,-1165,-33589,-416
C01072=-2535,57996,-1056,-1093,-33552,-193
C01073=-2535,57996,-2456,-1093,-33552,-193
C01074=-2537,58001,-2448,-1092,-33555,-193
C01075=-2543,57999,-2451,-1091,-33554,-190
C01076=-2548,57996,-2456,-1091,-33552,-188
C01077=-2552,57991,-2463,-1090,-33550,-187
C01078=-2555,57987,-2470,-1090,-33547,-185
C01079=-2560,57983,-2476,-1089,-33544,-183
C01080=-2565,57979,-2482,-1089,-33542,-181
C01081=-2569,57974,-2489,-1088,-33539,-180
C01082=-2573,57970,-2496,-1088,-33537,-178
C01083=-2578,57967,-2501,-1087,-33534,-176
C01084=-2583,57964,-2505,-1087,-33533,-174
C01085=-2588,57961,-2509,-1086,-33531,-171
C01086=-2594,57960,-2511,-1085,-33531,-169
C01087=-2600,57960,-2512,-1084,-33530,-167
C01088=-2606,57960,-2511,-1084,-33530,-164
C01089=-2612,57961,-2509,-1083,-33531,-162
C01090=-2618,57963,-2507,-1082,-33532,-160
C01091=-2623,57966,-2502,-1081,-33534,-158
C01092=-2628,57969,-2497,-1081,-33536,-156
C01093=-2633,57973,-2491,-1080,-33538,-154
C01094=-2636,57978,-2484,-1079,-33541,-153
C01095=-2640,57983,-2477,-1079,-33544,-151
C01096=-2642,57988,-2469,-1078,-33548,-150
C01097=-2646,57993,-2461,-1078,-33551,-149
C01098=-2649,57999,-2453,-1077,-33554,-148
C01099=-2648,58005,-2444,-1077,-33558,-148
C01100=-2649,58011,-2435,-1077,-33561,-148
C01101=-2655,58013,-2432,-1076,-33562,-145
C01102=-2660,58011,-2434,-1076,-33562,-143
C01103=-2663,58006,-2442,-1075,-33558,-142
C01104=-2663,58000,-2451,-1075,-33555,-142
C01105=-2662,57995,-2460,-1076,-33551,-142
C01106=-2659,57989,-2468,-1076,-33548,-143
C01107=-2655,57984,-2475,-1077,-33545,-145
C01108=-2653,57979,-2483,-1077,-33542,-146
C01109=-2650,57974,-2491,-1078,-33539,-147
C01110=-2646,57969,-2498,-1078,-33536,-148
C01111=-2642,57965,-2505,-1079,-33533,-150
C01112=-2637,57961,-2510,-1080,-33531,-152
C01113=-2633,57957,-2516,-1080,-33528,-154
C01114=-2628,57953,-2522,-1081,-33526,-156
C01115=-2622,57951,-2525,-1082,-33525,-158
C01116=-2617,57949,-2528,-1082,-33524,-160
C01117=-2610,57948,-2529,-1083,-33523,-162
C01118=-2604,57948,-2529,-1084,-33523,-165
C01119=-2598,57948,-2530,-1085,-33523,-168
C01120=-2592,57949,-2527,-1086,-33524,-170
C01121=-2587,57951,-2525,-1086,-33525,-172
C01122=-2581,57953,-2522,-1087,-33526,-174
C01123=-2576,57955,-2518,-1088,-33527,-176
C01124=-2571,57958,-2514,-1088,-33529,-179
C01125=-2566,57961,-2509,-1089,-33531,-181
C01126=-2561,57964,-2504,-1090,-33533,-183
C01127=-2556,57968,-2498,-1090,-33536,-184
C01128=-2552,57973,-2491,-1091,-33538,-186
C01129=-2548,57977,-2485,-1091,-33541,-188
C01130=-2543,57981,-2478,-1092,-33543,-190
C01131=-2539,57986,-2471,-1092,-33546,-191
C01132=-2537,57991,-2464,-1092,-33549,-193
C01133=-2535,57996,-2456,-1093,-33552,-193
C01134=-2535,57996,-1056,-1093,-33552,-193
C01135=-2619,57782,-1379,-1085,-33423,-157
C01136=-2619,57782,-2779,-1085,-33423,-157
C01137=-2609,57776,-2789,-1086,-33419,-161
C01138=-2598,57768,-2801,-1088,-33414,-165
C01139=-2588,57759,-2815,-1089,-33408,-169
C01140=-2578,57750,-2828,-1091,-33403,-173
C01141=-2568,57740,-2842,-1092,-33397,-177
C01142=-2557,57732,-2855,-1094,-33392,-181
C01143=-2546,57723,-2868,-1095,-33387,-185
C01144=-2535,57716,-2878,-1097,-33382,-190
C01145=-2525,57708,-2891,-1098,-33377,-194
C01146=-2513,57701,-2902,-1100,-33373,-198
C01147=-2502,57693,-2914,-1102,-33368,-203
C01148=-2492,57685,-2925,-1103,-33363,-207
C01149=-2481,57677,-2937,-1105,-33359,-211
C01150=-2470,57669,-2950,-1106,-33353,-215
C01151=-2459,57660,-2962,-1108,-33348,-220
C01152=-2449,57652,-2975,-1109,-33343,-224
C01153=-2438,57643,-2988,-1111,-33338,-228
C01154=-2427,57635,-3000,-1112,-33333,-232
C01155=-2417,57626,-3013,-1114,-33328,-236
C01156=-2421,57616,-3028,-1114,-33321,-235
C01157=-2430,57607,-3042,-1113,-33316,-231
C01158=-2440,57598,-3056,-1111,-33310,-226
C01159=-2450,57591,-3067,-1110,-33306,-222
C01160=-2461,57582,-3080,-1109,-33301,-218
C01161=-2471,57574,-3092,-1108,-33296,-214
C01162=-2482,57566,-3104,-1106,-33291,-209
C01163=-2493,57560,-3114,-1105,-33287,-205
C01164=-2504,57553,-3125,-1103,-33283,-200
C01165=-2516,57547,-3134,-1102,-33280,-195
C01166=-2527,57540,-3144,-1101,-33275,-191
C01167=-2538,57533,-3155,-1099,-33271,-186
C01168=-2550,57527,-3164,-1098,-33267,-182
C01169=-2560,57519,-3176,-1097,-33263,-177
C01170=-2571,57510,-3190,-1095,-33257,-173
C01171=-2582,57503,-3201,-1094,-33253,-169
C01172=-2592,57494,-3214,-1093,-33248,-165
C01173=-2602,57486,-3226,-1091,-33243,-160
C01174=-2609,57488,-3224,-1090,-33244,-157
C01175=-2611,57501,-3204,-1090,-33252,-157
C01176=-2611,57515,-3183,-1090,-33260,-157
C01177=-2609,57528,-3163,-1090,-33268,-158
C01178=-2610,57542,-3142,-1090,-33277,-158
C01179=-2611,57555,-3122,-1089,-33285,-158
C01180=-2610,57569,-3101,-1089,-33293,-158
C01181=-2611,57583,-3081,-1089,-33302,-158
C01182=-2611,57597,-3060,-1089,-33310,-158
C01183=-2612,57610,-3040,-1088,-33318,-158
C01184=-2613,57623,-3019,-1088,-33326,-157
C01185=-2614,57636,-3000,-1088,-33334,-157
C01186=-2614,57649,-2980,-1087,-33342,-157
C01187=-2616,57662,-2961,-1087,-33350,-157
C01188=-2616,57676,-2940,-1087,-33358,-157
C01189=-2616,57690,-2919,-1086,-33366,-157
C01190=-2617,57703,-2899,-1086,-33375,-157
C01191=-2618,57717,-2878,-1086,-33383,-157
C01192=-2617,57730,-2858,-1086,-33391,-157
C01193=-2618,57743,-2839,-1085,-33399,-157
C01194=-2618,57755,-2820,-1085,-33406,-157
C01195=-2618,57769,-2800,-1085,-33414,-157
C01196=-2619,57782,-2779,-1085,-33423,-157
C01197=-2619,57782,-1379,-1085,-33423,-157
C01198=-2636,57767,-1403,-1083,-33413,-150
C01199=-2636,57767,-2803,-1083,-33413,-150
C01200=-2631,57758,-2816,-1084,-33408,-152
C01201=-2629,57744,-2837,-1084,-33400,-153
C01202=-2629,57730,-2859,-1084,-33391,-152
C01203=-2629,57716,-2880,-1084,-33382,-152
C01204=-2628,57702,-2901,-1085,-33374,-152
C01205=-2627,57688,-2922,-1085,-33365,-153
C01206=-2626,57674,-2943,-1085,-33357,-153
C01207=-2625,57660,-2964,-1086,-33349,-153
C01208=-2625,57646,-2985,-1086,-33340,-153
C01209=-2624,57632,-3006,-1086,-33332,-153
C01210=-2623,57618,-3027,-1087,-33323,-153
C01211=-2623,57605,-3048,-1087,-33315,-153
C01212=-2622,57591,-3069,-1087,-33306,-153
C01213=-2622,57576,-3090,-1087,-33298,-153
C01214=-2622,57562,-3112,-1088,-33289,-153
C01215=-2620,57549,-3132,-1088,-33281,-154
C01216=-2621,57534,-3154,-1088,-33272,-153
C01217=-2621,57520,-3176,-1088,-33263,-153
C01218=-2621,57506,-3196,-1089,-33255,-153
C01219=-2620,57492,-3217,-1089,-33247,-153
C01220=-2623,57480,-3236,-1089,-33239,-152
C01221=-2634,57487,-3226,-1087,-33243,-147
C01222=-2646,57493,-3216,-1085,-33247,-143
C01223=-2658,57501,-3204,-1084,-33252,-138
C01224=-2670,57507,-3196,-1082,-33256,-133
C01225=-2682,57513,-3186,-1080,-33259,-129
C01226=-2694,57519,-3178,-1079,-33263,-124
C01227=-2707,57524,-3171,-1077,-33266,-119
C01228=-2719,57530,-3162,-1075,-33270,-114
C01229=-2732,57534,-3155,-1073,-33272,-109
C01230=-2744,57540,-3146,-1072,-33276,-104
C01231=-2757,57546,-3137,-1070,-33280,-99
C01232=-2769,57552,-3128,-1068,-33283,-94
C01233=-2781,57558,-3120,-1067,-33287,-89
C01234=-2793,57564,-3111,-1065,-33291,-85
C01235=-2805,57570,-3102,-1063,-33294,-80
C01236=-2817,57577,-3091,-1061,-33298,-75
C01237=-2829,57584,-3081,-1060,-33303,-71
C01238=-2840,57592,-3069,-1058,-33308,-66
C01239=-2849,57600,-3057,-1057,-33313,-63
C01240=-2838,57609,-3043,-1058,-33318,-67
C01241=-2828,57618,-3030,-1059,-33323,-71
C01242=-2818,57627,-3017,-1061,-33328,-75
C01243=-2807,57635,-3004,-1062,-33333,-80
C01244=-2796,57643,-2992,-1063,-33338,-84
C01245=-2785,57651,-2979,-1065,-33343,-89
C01246=-2774,57658,-2969,-1066,-33347,-93
C01247=-2762,57665,-2958,-1067,-33352,-98
C01248=-2751,57673,-2947,-1069,-33356,-103
C01249=-2740,57680,-2935,-1070,-33361,-107
C01250=-2729,57689,-2922,-1072,-33366,-112
C01251=-2718,57696,-2911,-1073,-33370,-117
C01252=-2707,57705,-2897,-1074,-33376,-121
C01253=-2695,57713,-2886,-1076,-33380,-126
C01254=-2685,57721,-2873,-1077,-33386,-130
C01255=-2674,57730,-2860,-1078,-33391,-134
C01256=-2665,57739,-2845,-1079,-33396,-138
C01257=-2655,57748,-2832,-1080,-33402,-142
C01258=-2644,57756,-2819,-1082,-33407,-147
C01259=-2636,57767,-2803,-1083,-33413,-150
C01260=-2636,57767,-1403,-1083,-33413,-150
C01261=-1285,57892,-1195,-1260,-33491,-694
C01262=-1285,57892,-2595,-1260,-33491,-694
C01263=-1281,57890,-2598,-1260,-33489,-695
C01264=-1277,57889,-2600,-1261,-33489,-697
C01265=-1273,57891,-2596,-1261,-33490,-698
C01266=-1272,57895,-2590,-1261,-33493,-699
C01267=-1272,57900,-2583,-1261,-33496,-699
C01268=-1274,57904,-2577,-1261,-33498,-698
C01269=-1275,57908,-2571,-1261,-33501,-698
C01270=-1277,57912,-2564,-1260,-33503,-697
C01271=-1278,57916,-2558,-1260,-33506,-697
C01272=-1280,57920,-2552,-1260,-33508,-696
C01273=-1281,57925,-2545,-1260,-33511,-696
C01274=-1281,57929,-2538,-1259,-33514,-696
C01275=-1282,57933,-2532,-1259,-33516,-695
C01276=-1283,57938,-2525,-1259,-33519,-695
C01277=-1284,57942,-2519,-1259,-33522,-695
C01278=-1285,57946,-2512,-1259,-33524,-694
C01279=-1286,57951,-2505,-1258,-33527,-694
C01280=-1287,57955,-2499,-1258,-33530,-694
C01281=-1288,57959,-2493,-1258,-33532,-693
C01282=-1290,57963,-2486,-1258,-33535,-693
C01283=-1291,57968,-2480,-1257,-33537,-692
C01284=-1292,57972,-2473,-1257,-33540,-692
C01285=-1293,57976,-2467,-1257,-33543,-692
C01286=-1294,57981,-2460,-1257,-33545,-691
C01287=-1295,57985,-2454,-1257,-33548,-691
C01288=-1296,57989,-2447,-1256,-33551,-690
C01289=-1297,57993,-2441,-1256,-33553,-690
C01290=-1298,57998,-2434,-1256,-33556,-690
C01291=-1300,58002,-2428,-1256,-33559,-689
C01292=-1302,58006,-2422,-1255,-33561,-689
C01293=-1304,58010,-2416,-1255,-33563,-688
C01294=-1308,58011,-2414,-1254,-33564,-686
C01295=-1311,58008,-2419,-1254,-33562,-685
C01296=-1312,58004,-2425,-1254,-33560,-684
C01297=-1310,58000,-2431,-1254,-33557,-685
C01298=-1308,57996,-2438,-1255,-33555,-686
C01299=-1307,57991,-2444,-1255,-33552,-686
C01300=-1306,57987,-2450,-1255,-33549,-687
C01301=-1305,57983,-2457,-1255,-33547,-687
C01302=-1304,57978,-2464,-1256,-33544,-687
C01303=-1303,57974,-2470,-1256,-33541,-688
C01304=-1302,57970,-2477,-1256,-33539,-688
C01305=-1301,57965,-2483,-1256,-33536,-688
C01306=-1300,57961,-2490,-1256,-33533,-688
C01307=-1300,57957,-2497,-1257,-33531,-689
C01308=-1298,57953,-2503,-1257,-33528,-689
C01309=-1296,57949,-2509,-1257,-33526,-690
C01310=-1295,57944,-2515,-1257,-33523,-690
C01311=-1294,57940,-2522,-1258,-33520,-691
C01312=-1293,57936,-2529,-1258,-33518,-691
C01313=-1293,57931,-2536,-1258,-33515,-691
C01314=-1292,57927,-2542,-1258,-33512,-691
C01315=-1291,57923,-2549,-1258,-33510,-692
C01316=-1289,57918,-2555,-1259,-33507,-692
C01317=-1288,57914,-2561,-1259,-33504,-693
C01318=-1287,57910,-2568,-1259,-33502,-693
C01319=-1286,57905,-2574,-1259,-33499,-693
C01320=-1286,57901,-2581,-1259,-33496,-693
C01321=-1285,57897,-2588,-1260,-33494,-694
C01322=-1285,57892,-2595,-1260,-33491,-694
C01323=-1285,57892,-1195,-1260,-33491,-694
C01324=-1239,57891,-1195,-1266,-33490,-712
C01325=-1239,57891,-2595,-1266,-33490,-712
C01326=-1235,57879,-2615,-1266,-33482,-713
C01327=-1226,57868,-2631,-1268,-33476,-717
C01328=-1214,57861,-2641,-1270,-33472,-722
C01329=-1200,57859,-2644,-1271,-33471,-727
C01330=-1186,57861,-2641,-1273,-33472,-733
C01331=-1174,57866,-2633,-1275,-33475,-738
C01332=-1162,57873,-2623,-1276,-33479,-742
C01333=-1153,57882,-2608,-1277,-33485,-746
C01334=-1146,57893,-2591,-1278,-33492,-749
C01335=-1142,57906,-2572,-1278,-33499,-751
C01336=-1143,57919,-2551,-1278,-33508,-751
C01337=-1150,57931,-2533,-1277,-33515,-748
C01338=-1161,57939,-2521,-1275,-33520,-744
C01339=-1173,57946,-2511,-1273,-33524,-739
C01340=-1187,57949,-2507,-1272,-33526,-734
C01341=-1201,57951,-2503,-1270,-33528,-728
C01342=-1215,57953,-2501,-1268,-33529,-723
C01343=-1229,57955,-2498,-1266,-33530,-717
C01344=-1242,57960,-2491,-1264,-33533,-712
C01345=-1252,57969,-2478,-1263,-33538,-708
C01346=-1255,57982,-2457,-1262,-33546,-707
C01347=-1248,57993,-2440,-1263,-33554,-710
C01348=-1237,58001,-2428,-1264,-33558,-714
C01349=-1224,58004,-2423,-1266,-33560,-720
C01350=-1210,58003,-2425,-1268,-33559,-725
C01351=-1197,57998,-2433,-1269,-33556,-730
C01352=-1187,57988,-2447,-1271,-33550,-734
C01353=-1177,57978,-2463,-1272,-33544,-738
C01354=-1176,57987,-2448,-1272,-33550,-739
C01355=-1182,57999,-2430,-1271,-33557,-736
C01356=-1194,58008,-2417,-1270,-33562,-732
C01357=-1206,58013,-2409,-1268,-33566,-727
C01358=-1220,58016,-2405,-1266,-33567,-721
C01359=-1234,58015,-2407,-1264,-33567,-716
C01360=-1246,58009,-2416,-1263,-33563,-711
C01361=-1257,58000,-2429,-1261,-33558,-707
C01362=-1264,57990,-2446,-1261,-33551,-703
C01363=-1266,57976,-2467,-1261,-33543,-702
C01364=-1261,57963,-2486,-1261,-33535,-704
C01365=-1252,57953,-2501,-1263,-33529,-708
C01366=-1239,57948,-2509,-1265,-33526,-713
C01367=-1225,57946,-2512,-1267,-33524,-718
C01368=-1211,57943,-2516,-1268,-33522,-724
C01369=-1197,57942,-2517,-1270,-33522,-730
C01370=-1183,57939,-2522,-1272,-33520,-735
C01371=-1170,57934,-2528,-1274,-33517,-740
C01372=-1159,57927,-2540,-1276,-33513,-745
C01373=-1152,57915,-2558,-1277,-33505,-747
C01374=-1153,57901,-2579,-1277,-33497,-747
C01375=-1160,57890,-2596,-1276,-33490,-744
C01376=-1170,57881,-2610,-1275,-33484,-740
C01377=-1182,57875,-2620,-1274,-33480,-735
C01378=-1194,57870,-2628,-1272,-33477,-730
C01379=-1208,57870,-2628,-1270,-33477,-724
C01380=-1220,57876,-2618,-1268,-33481,-719
C01381=-1228,57887,-2602,-1267,-33488,-716
C01382=-1234,57899,-2583,-1266,-33495,-714
C01383=-1237,57912,-2563,-1266,-33503,-713
C01384=-1242,57905,-2575,-1265,-33499,-711
C01385=-1239,57891,-2595,-1266,-33490,-712
C01386=-1239,57891,-1195,-1266,-33490,-712
C01387=-1074,57925,-1141,-1287,-33512,-779
C01388=-1074,57925,-2541,-1287,-33512,-779
C01389=-1067,57924,-2543,-1288,-33511,-782
C01390=-1063,57931,-2533,-1288,-33515,-783
C01391=-1060,57937,-2523,-1289,-33519,-785
C01392=-1058,57944,-2512,-1289,-33524,-785
C01393=-1054,57951,-2502,-1289,-33528,-787
C01394=-1050,57958,-2491,-1289,-33532,-789
C01395=-1047,57964,-2481,-1290,-33536,-790
C01396=-1043,57971,-2471,-1290,-33540,-792
C01397=-1038,57977,-2462,-1291,-33544,-794
C01398=-1034,57984,-2451,-1291,-33548,-796
C01399=-1029,57990,-2442,-1292,-33552,-798
C01400=-1026,57997,-2431,-1292,-33556,-799
C01401=-1023,58004,-2420,-1292,-33561,-800
C01402=-1021,58011,-2409,-1292,-33565,-801
C01403=-1018,58019,-2398,-1293,-33570,-802
C01404=-1017,58026,-2386,-1293,-33575,-803
C01405=-1017,58035,-2373,-1292,-33580,-803
C01406=-1018,58043,-2361,-1292,-33585,-803
C01407=-1019,58050,-2349,-1292,-33589,-803
C01408=-1023,58057,-2339,-1291,-33594,-801
C01409=-1029,58062,-2332,-1290,-33597,-799
C01410=-1037,58065,-2327,-1289,-33599,-796
C01411=-1045,58066,-2325,-1288,-33599,-793
C01412=-1053,58067,-2325,-1287,-33600,-789
C01413=-1061,58065,-2328,-1286,-33598,-786
C01414=-1068,58062,-2332,-1285,-33597,-783
C01415=-1076,58060,-2335,-1284,-33595,-780
C01416=-1083,58058,-2339,-1283,-33594,-777
C01417=-1090,58055,-2344,-1282,-33592,-774
C01418=-1096,58050,-2352,-1282,-33589,-772
C01419=-1102,58044,-2361,-1281,-33585,-769
C01420=-1101,58036,-2373,-1281,-33580,-770
C01421=-1093,58033,-2377,-1282,-33579,-773
C01422=-1090,58040,-2367,-1283,-33583,-774
C01423=-1085,58045,-2359,-1283,-33586,-776
C01424=-1078,58049,-2353,-1284,-33588,-779
C01425=-1070,58052,-2348,-1285,-33590,-782
C01426=-1063,58054,-2345,-1286,-33592,-785
C01427=-1056,58056,-2341,-1287,-33593,-788
C01428=-1047,58057,-2340,-1288,-33593,-791
C01429=-1040,58054,-2343,-1289,-33592,-794
C01430=-1033,58051,-2349,-1290,-33590,-797
C01431=-1029,58044,-2360,-1291,-33585,-799
C01432=-1027,58036,-2371,-1291,-33580,-799
C01433=-1028,58028,-2384,-1291,-33576,-799
C01434=-1029,58020,-2396,-1291,-33571,-798
C01435=-1031,58013,-2407,-1291,-33566,-797
C01436=-1034,58005,-2418,-1291,-33562,-796
C01437=-1037,57999,-2428,-1290,-33557,-795
C01438=-1041,57992,-2438,-1290,-33553,-793
C01439=-1045,57986,-2449,-1290,-33549,-791
C01440=-1050,57979,-2458,-1289,-33545,-789
C01441=-1054,57973,-2468,-1289,-33541,-787
C01442=-1058,57966,-2479,-1288,-33537,-786
C01443=-1061,57959,-2489,-1288,-33533,-784
C01444=-1065,57953,-2499,-1288,-33529,-783
C01445=-1068,57946,-2510,-1287,-33524,-781
C01446=-1072,57939,-2520,-1287,-33520,-780
C01447=-1075,57932,-2531,-1287,-33516,-779
C01448=-1074,57925,-2541,-1287,-33512,-779
C01449=-1074,57925,-1141,-1287,-33512,-779
C01450=-1060,57864,-1234,-1290,-33474,-783
C01451=-1060,57864,-2634,-1290,-33474,-783
C01452=-1061,57863,-2635,-1290,-33473,-783
C01453=-1062,57863,-2637,-1290,-33473,-783
C01454=-1062,57862,-2638,-1290,-33472,-782
C01455=-1063,57861,-2639,-1289,-33472,-782
C01456=-1064,57860,-2640,-1289,-33471,-782
C01457=-1065,57859,-2641,-1289,-33471,-781
C01458=-1066,57859,-2643,-1289,-33470,-781
C01459=-1066,57858,-2644,-1289,-33470,-781
C01460=-1067,57857,-2645,-1289,-33469,-781
C01461=-1068,57856,-2647,-1289,-33469,-780
C01462=-1069,57855,-2648,-1289,-33468,-780
C01463=-1070,57854,-2649,-1289,-33468,-779
C01464=-1070,57854,-2650,-1289,-33467,-779
C01465=-1070,57852,-2652,-1289,-33467,-779
C01466=-1070,57851,-2654,-1289,-33466,-779
C01467=-1069,57850,-2655,-1289,-33465,-779
C01468=-1069,57849,-2657,-1289,-33465,-779
C01469=-1069,57848,-2659,-1289,-33464,-780
C01470=-1068,57847,-2660,-1289,-33463,-780
C01471=-1068,57846,-2662,-1289,-33463,-780
C01472=-1067,57846,-2663,-1289,-33462,-780
C01473=-1066,57845,-2663,-1289,-33462,-781
C01474=-1065,57845,-2664,-1290,-33462,-781
C01475=-1064,57844,-2664,-1290,-33462,-782
C01476=-1063,57844,-2665,-1290,-33461,-782
C01477=-1062,57843,-2666,-1290,-33461,-782
C01478=-1061,57843,-2666,-1290,-33461,-783
C01479=-1060,57844,-2665,-1290,-33461,-783
C01480=-1058,57844,-2665,-1290,-33461,-784
C01481=-1058,57845,-2664,-1291,-33462,-784
C01482=-1057,57846,-2662,-1291,-33462,-784
C01483=-1056,57846,-2661,-1291,-33463,-785
C01484=-1055,57847,-2661,-1291,-33463,-785
C01485=-1054,57847,-2660,-1291,-33463,-786
C01486=-1053,57848,-2659,-1291,-33464,-786
C01487=-1052,57848,-2658,-1291,-33464,-786
C01488=-1051,57849,-2657,-1291,-33464,-787
C01489=-1050,57850,-2656,-1291,-33465,-787
C01490=-1050,57851,-2654,-1291,-33466,-787
C01491=-1049,57852,-2653,-1292,-33466,-788
C01492=-1048,57852,-2652,-1292,-33467,-788
C01493=-1047,57853,-2651,-1292,-33467,-788
C01494=-1046,57854,-2649,-1292,-33468,-789
C01495=-1046,57855,-2648,-1292,-33468,-789
C01496=-1046,57856,-2646,-1292,-33469,-789
C01497=-1047,57857,-2645,-1292,-33469,-789
C01498=-1047,57858,-2643,-1292,-33470,-789
C01499=-1048,57858,-2643,-1292,-33470,-788
C01500=-1049,57859,-2642,-1291,-33471,-788
C01501=-1050,57859,-2642,-1291,-33471,-787
C01502=-1051,57859,-2642,-1291,-33471,-787
C01503=-1053,57859,-2641,-1291,-33471,-786
C01504=-1054,57860,-2641,-1291,-33471,-786
C01505=-1055,57860,-2640,-1291,-33471,-785
C01506=-1056,57861,-2639,-1290,-33472,-785
C01507=-1056,57862,-2638,-1290,-33472,-785
C01508=-1057,57863,-2636,-1290,-33473,-785
C01509=-1058,57864,-2635,-1290,-33474,-784
C01510=-1059,57864,-2634,-1290,-33474,-784
C01511=-1060,57864,-2634,-1290,-33474,-783
C01512=-1060,57864,-1234,-1290,-33474,-783
C01513=-1302,58038,-973,-1255,-33581,-689
C01514=-1302,58038,-2373,-1255,-33581,-689
C01515=-1302,58038,-2373,-1255,-33581,-689
C01516=-1302,58038,-2373,-1255,-33581,-689
C01517=-1301,58038,-2372,-1255,-33581,-689
C01518=-1301,58039,-2372,-1255,-33581,-689
C01519=-1301,58039,-2371,-1255,-33582,-689
C01520=-1301,58040,-2370,-1255,-33582,-689
C01521=-1301,58040,-2369,-1255,-33582,-689
C01522=-1301,58041,-2369,-1255,-33583,-689
C01523=-1300,58041,-2368,-1255,-33583,-690
C01524=-1300,58042,-2367,-1255,-33583,-690
C01525=-1300,58042,-2367,-1255,-33583,-690
C01526=-1300,58043,-2366,-1255,-33584,-690
C01527=-1300,58043,-2365,-1255,-33584,-690
C01528=-1300,58044,-2364,-1255,-33584,-690
C01529=-1300,58044,-2363,-1255,-33585,-690
C01530=-1301,58045,-2363,-1255,-33585,-689
C01531=-1301,58045,-2362,-1255,-33585,-689
C01532=-1302,58045,-2362,-1255,-33585,-689
C01533=-1302,58046,-2361,-1255,-33586,-689
C01534=-1302,58046,-2361,-1255,-33586,-689
C01535=-1303,58046,-2360,-1254,-33586,-689
C01536=-1303,58047,-2360,-1254,-33586,-688
C01537=-1304,58047,-2360,-1254,-33586,-688
C01538=-1304,58047,-2360,-1254,-33586,-688
C01539=-1305,58047,-2360,-1254,-33586,-688
C01540=-1305,58047,-2360,-1254,-33586,-688
C01541=-1306,58047,-2359,-1254,-33586,-687
C01542=-1306,58047,-2359,-1254,-33586,-687
C01543=-1307,58047,-2359,-1254,-33586,-687
C01544=-1307,58047,-2359,-1254,-33586,-687
C01545=-1308,58047,-2360,-1254,-33586,-687
C01546=-1308,58046,-2360,-1254,-33586,-686
C01547=-1309,58046,-2361,-1254,-33586,-686
C01548=-1309,58046,-2362,-1254,-33586,-686
C01549=-1309,58045,-2362,-1254,-33585,-686
C01550=-1310,58045,-2363,-1254,-33585,-686
C01551=-1310,58044,-2363,-1254,-33585,-686
C01552=-1310,58044,-2364,-1254,-33585,-686
C01553=-1310,58043,-2365,-1254,-33584,-686
C01554=-1310,58043,-2365,-1254,-33584,-686
C01555=-1310,58042,-2366,-1254,-33584,-686
C01556=-1310,58042,-2367,-1254,-33583,-686
C01557=-1310,58041,-2368,-1254,-33583,-686
C01558=-1310,58041,-2368,-1254,-33583,-686
C01559=-1309,58041,-2369,-1254,-33583,-686
C01560=-1309,58041,-2369,-1254,-33583,-686
C01561=-1308,58040,-2369,-1254,-33582,-686
C01562=-1308,58040,-2370,-1254,-33582,-686
C01563=-1308,58040,-2370,-1254,-33582,-687
C01564=-1307,58039,-2371,-1254,-33582,-687
C01565=-1307,58039,-2372,-1254,-33581,-687
C01566=-1306,58039,-2372,-1254,-33581,-687
C01567=-1306,58038,-2373,-1254,-33581,-687
C01568=-1306,58038,-2373,-1254,-33581,-687
C01569=-1305,58038,-2373,-1254,-33581,-688
C01570=-1305,58038,-2373,-1254,-33581,-688
C01571=-1304,58038,-2373,-1254,-33581,-688
C01572=-1304,58038,-2373,-1255,-33581,-688
C01573=-1303,58038,-2373,-1255,-33581,-688
C01574=-1302,58038,-2373,-1255,-33581,-689
C01575=-1302,58038,-973,-1255,-33581,-689
//INST
///DATE 2026/04/22 18:45
///ATTR SC,RW
///GROUP1 RB1
NOP
MOVJ C00000 VJ=0.78
MOVJ C00001 VJ=0.78
MOVJ C00002 VJ=0.78
MOVL C00003 V=8.0
MOVL C00004 V=8.0
MOVL C00005 V=8.0
MOVL C00006 V=8.0
MOVL C00007 V=8.0
MOVL C00008 V=8.0
MOVL C00009 V=8.0
MOVL C00010 V=8.0
MOVL C00011 V=8.0
MOVL C00012 V=8.0
MOVL C00013 V=8.0
MOVL C00014 V=8.0
MOVL C00015 V=8.0
MOVL C00016 V=8.0
MOVL C00017 V=8.0
MOVL C00018 V=8.0
MOVL C00019 V=8.0
MOVL C00020 V=8.0
MOVL C00021 V=8.0
MOVL C00022 V=8.0
MOVL C00023 V=8.0
MOVL C00024 V=8.0
MOVL C00025 V=8.0
MOVL C00026 V=8.0
MOVL C00027 V=8.0
MOVL C00028 V=8.0
MOVL C00029 V=8.0
MOVL C00030 V=8.0
MOVL C00031 V=8.0
MOVL C00032 V=8.0
MOVL C00033 V=8.0
MOVL C00034 V=8.0
MOVL C00035 V=8.0
MOVL C00036 V=8.0
MOVL C00037 V=8.0
MOVL C00038 V=8.0
MOVL C00039 V=8.0
MOVL C00040 V=8.0
MOVL C00041 V=8.0
MOVL C00042 V=8.0
MOVL C00043 V=8.0
MOVL C00044 V=8.0
MOVL C00045 V=8.0
MOVL C00046 V=8.0
MOVL C00047 V=8.0
MOVL C00048 V=8.0
MOVL C00049 V=8.0
MOVL C00050 V=8.0
MOVL C00051 V=8.0
MOVL C00052 V=8.0
MOVL C00053 V=8.0
MOVL C00054 V=8.0
MOVL C00055 V=8.0
MOVL C00056 V=8.0
MOVL C00057 V=8.0
MOVL C00058 V=8.0
MOVL C00059 V=8.0
MOVL C00060 V=8.0
MOVL C00061 V=8.0
MOVL C00062 V=8.0
MOVJ C00063 VJ=0.78
MOVJ C00064 VJ=0.78
MOVJ C00065 VJ=0.78
MOVL C00066 V=8.0
MOVL C00067 V=8.0
MOVL C00068 V=8.0
MOVL C00069 V=8.0
MOVL C00070 V=8.0
MOVL C00071 V=8.0
MOVL C00072 V=8.0
MOVL C00073 V=8.0
MOVL C00074 V=8.0
MOVL C00075 V=8.0
MOVL C00076 V=8.0
MOVL C00077 V=8.0
MOVL C00078 V=8.0
MOVL C00079 V=8.0
MOVL C00080 V=8.0
MOVL C00081 V=8.0
MOVL C00082 V=8.0
MOVL C00083 V=8.0
MOVL C00084 V=8.0
MOVL C00085 V=8.0
MOVL C00086 V=8.0
MOVL C00087 V=8.0
MOVL C00088 V=8.0
MOVL C00089 V=8.0
MOVL C00090 V=8.0
MOVL C00091 V=8.0
MOVL C00092 V=8.0
MOVL C00093 V=8.0
MOVL C00094 V=8.0
MOVL C00095 V=8.0
MOVL C00096 V=8.0
MOVL C00097 V=8.0
MOVL C00098 V=8.0
MOVL C00099 V=8.0
MOVL C00100 V=8.0
MOVL C00101 V=8.0
MOVL C00102 V=8.0
MOVL C00103 V=8.0
MOVL C00104 V=8.0
MOVL C00105 V=8.0
MOVL C00106 V=8.0
MOVL C00107 V=8.0
MOVL C00108 V=8.0
MOVL C00109 V=8.0
MOVL C00110 V=8.0
MOVL C00111 V=8.0
MOVL C00112 V=8.0
MOVL C00113 V=8.0
MOVL C00114 V=8.0
MOVL C00115 V=8.0
MOVL C00116 V=8.0
MOVL C00117 V=8.0
MOVL C00118 V=8.0
MOVL C00119 V=8.0
MOVL C00120 V=8.0
MOVL C00121 V=8.0
MOVL C00122 V=8.0
MOVL C00123 V=8.0
MOVL C00124 V=8.0
MOVL C00125 V=8.0
MOVJ C00126 VJ=0.78
MOVJ C00127 VJ=0.78
MOVJ C00128 VJ=0.78
MOVL C00129 V=8.0
MOVL C00130 V=8.0
MOVL C00131 V=8.0
MOVL C00132 V=8.0
MOVL C00133 V=8.0
MOVL C00134 V=8.0
MOVL C00135 V=8.0
MOVL C00136 V=8.0
MOVL C00137 V=8.0
MOVL C00138 V=8.0
MOVL C00139 V=8.0
MOVL C00140 V=8.0
MOVL C00141 V=8.0
MOVL C00142 V=8.0
MOVL C00143 V=8.0
MOVL C00144 V=8.0
MOVL C00145 V=8.0
MOVL C00146 V=8.0
MOVL C00147 V=8.0
MOVL C00148 V=8.0
MOVL C00149 V=8.0
MOVL C00150 V=8.0
MOVL C00151 V=8.0
MOVL C00152 V=8.0
MOVL C00153 V=8.0
MOVL C00154 V=8.0
MOVL C00155 V=8.0
MOVL C00156 V=8.0
MOVL C00157 V=8.0
MOVL C00158 V=8.0
MOVL C00159 V=8.0
MOVL C00160 V=8.0
MOVL C00161 V=8.0
MOVL C00162 V=8.0
MOVL C00163 V=8.0
MOVL C00164 V=8.0
MOVL C00165 V=8.0
MOVL C00166 V=8.0
MOVL C00167 V=8.0
MOVL C00168 V=8.0
MOVL C00169 V=8.0
MOVL C00170 V=8.0
MOVL C00171 V=8.0
MOVL C00172 V=8.0
MOVL C00173 V=8.0
MOVL C00174 V=8.0
MOVL C00175 V=8.0
MOVL C00176 V=8.0
MOVL C00177 V=8.0
MOVL C00178 V=8.0
MOVL C00179 V=8.0
MOVL C00180 V=8.0
MOVL C00181 V=8.0
MOVL C00182 V=8.0
MOVL C00183 V=8.0
MOVL C00184 V=8.0
MOVL C00185 V=8.0
MOVL C00186 V=8.0
MOVL C00187 V=8.0
MOVL C00188 V=8.0
MOVJ C00189 VJ=0.78
MOVJ C00190 VJ=0.78
MOVJ C00191 VJ=0.78
MOVL C00192 V=8.0
MOVL C00193 V=8.0
MOVL C00194 V=8.0
MOVL C00195 V=8.0
MOVL C00196 V=8.0
MOVL C00197 V=8.0
MOVL C00198 V=8.0
MOVL C00199 V=8.0
MOVL C00200 V=8.0
MOVL C00201 V=8.0
MOVL C00202 V=8.0
MOVL C00203 V=8.0
MOVL C00204 V=8.0
MOVL C00205 V=8.0
MOVL C00206 V=8.0
MOVL C00207 V=8.0
MOVL C00208 V=8.0
MOVL C00209 V=8.0
MOVL C00210 V=8.0
MOVL C00211 V=8.0
MOVL C00212 V=8.0
MOVL C00213 V=8.0
MOVL C00214 V=8.0
MOVL C00215 V=8.0
MOVL C00216 V=8.0
MOVL C00217 V=8.0
MOVL C00218 V=8.0
MOVL C00219 V=8.0
MOVL C00220 V=8.0
MOVL C00221 V=8.0
MOVL C00222 V=8.0
MOVL C00223 V=8.0
MOVL C00224 V=8.0
MOVL C00225 V=8.0
MOVL C00226 V=8.0
MOVL C00227 V=8.0
MOVL C00228 V=8.0
MOVL C00229 V=8.0
MOVL C00230 V=8.0
MOVL C00231 V=8.0
MOVL C00232 V=8.0
MOVL C00233 V=8.0
MOVL C00234 V=8.0
MOVL C00235 V=8.0
MOVL C00236 V=8.0
MOVL C00237 V=8.0
MOVL C00238 V=8.0
MOVL C00239 V=8.0
MOVL C00240 V=8.0
MOVL C00241 V=8.0
MOVL C00242 V=8.0
MOVL C00243 V=8.0
MOVL C00244 V=8.0
MOVL C00245 V=8.0
MOVL C00246 V=8.0
MOVL C00247 V=8.0
MOVL C00248 V=8.0
MOVL C00249 V=8.0
MOVL C00250 V=8.0
MOVL C00251 V=8.0
MOVJ C00252 VJ=0.78
MOVJ C00253 VJ=0.78
MOVJ C00254 VJ=0.78
MOVL C00255 V=8.0
MOVL C00256 V=8.0
MOVL C00257 V=8.0
MOVL C00258 V=8.0
MOVL C00259 V=8.0
MOVL C00260 V=8.0
MOVL C00261 V=8.0
MOVL C00262 V=8.0
MOVL C00263 V=8.0
MOVL C00264 V=8.0
MOVL C00265 V=8.0
MOVL C00266 V=8.0
MOVL C00267 V=8.0
MOVL C00268 V=8.0
MOVL C00269 V=8.0
MOVL C00270 V=8.0
MOVL C00271 V=8.0
MOVL C00272 V=8.0
MOVL C00273 V=8.0
MOVL C00274 V=8.0
MOVL C00275 V=8.0
MOVL C00276 V=8.0
MOVL C00277 V=8.0
MOVL C00278 V=8.0
MOVL C00279 V=8.0
MOVL C00280 V=8.0
MOVL C00281 V=8.0
MOVL C00282 V=8.0
MOVL C00283 V=8.0
MOVL C00284 V=8.0
MOVL C00285 V=8.0
MOVL C00286 V=8.0
MOVL C00287 V=8.0
MOVL C00288 V=8.0
MOVL C00289 V=8.0
MOVL C00290 V=8.0
MOVL C00291 V=8.0
MOVL C00292 V=8.0
MOVL C00293 V=8.0
MOVL C00294 V=8.0
MOVL C00295 V=8.0
MOVL C00296 V=8.0
MOVL C00297 V=8.0
MOVL C00298 V=8.0
MOVL C00299 V=8.0
MOVL C00300 V=8.0
MOVL C00301 V=8.0
MOVL C00302 V=8.0
MOVL C00303 V=8.0
MOVL C00304 V=8.0
MOVL C00305 V=8.0
MOVL C00306 V=8.0
MOVL C00307 V=8.0
MOVL C00308 V=8.0
MOVL C00309 V=8.0
MOVL C00310 V=8.0
MOVL C00311 V=8.0
MOVL C00312 V=8.0
MOVL C00313 V=8.0
MOVL C00314 V=8.0
MOVJ C00315 VJ=0.78
MOVJ C00316 VJ=0.78
MOVJ C00317 VJ=0.78
MOVL C00318 V=8.0
MOVL C00319 V=8.0
MOVL C00320 V=8.0
MOVL C00321 V=8.0
MOVL C00322 V=8.0
MOVL C00323 V=8.0
MOVL C00324 V=8.0
MOVL C00325 V=8.0
MOVL C00326 V=8.0
MOVL C00327 V=8.0
MOVL C00328 V=8.0
MOVL C00329 V=8.0
MOVL C00330 V=8.0
MOVL C00331 V=8.0
MOVL C00332 V=8.0
MOVL C00333 V=8.0
MOVL C00334 V=8.0
MOVL C00335 V=8.0
MOVL C00336 V=8.0
MOVL C00337 V=8.0
MOVL C00338 V=8.0
MOVL C00339 V=8.0
MOVL C00340 V=8.0
MOVL C00341 V=8.0
MOVL C00342 V=8.0
MOVL C00343 V=8.0
MOVL C00344 V=8.0
MOVL C00345 V=8.0
MOVL C00346 V=8.0
MOVL C00347 V=8.0
MOVL C00348 V=8.0
MOVL C00349 V=8.0
MOVL C00350 V=8.0
MOVL C00351 V=8.0
MOVL C00352 V=8.0
MOVL C00353 V=8.0
MOVL C00354 V=8.0
MOVL C00355 V=8.0
MOVL C00356 V=8.0
MOVL C00357 V=8.0
MOVL C00358 V=8.0
MOVL C00359 V=8.0
MOVL C00360 V=8.0
MOVL C00361 V=8.0
MOVL C00362 V=8.0
MOVL C00363 V=8.0
MOVL C00364 V=8.0
MOVL C00365 V=8.0
MOVL C00366 V=8.0
MOVL C00367 V=8.0
MOVL C00368 V=8.0
MOVL C00369 V=8.0
MOVL C00370 V=8.0
MOVL C00371 V=8.0
MOVL C00372 V=8.0
MOVL C00373 V=8.0
MOVL C00374 V=8.0
MOVL C00375 V=8.0
MOVL C00376 V=8.0
MOVL C00377 V=8.0
MOVJ C00378 VJ=0.78
MOVJ C00379 VJ=0.78
MOVJ C00380 VJ=0.78
MOVL C00381 V=8.0
MOVL C00382 V=8.0
MOVL C00383 V=8.0
MOVL C00384 V=8.0
MOVL C00385 V=8.0
MOVL C00386 V=8.0
MOVL C00387 V=8.0
MOVL C00388 V=8.0
MOVL C00389 V=8.0
MOVL C00390 V=8.0
MOVL C00391 V=8.0
MOVL C00392 V=8.0
MOVL C00393 V=8.0
MOVL C00394 V=8.0
MOVL C00395 V=8.0
MOVL C00396 V=8.0
MOVL C00397 V=8.0
MOVL C00398 V=8.0
MOVL C00399 V=8.0
MOVL C00400 V=8.0
MOVL C00401 V=8.0
MOVL C00402 V=8.0
MOVL C00403 V=8.0
MOVL C00404 V=8.0
MOVL C00405 V=8.0
MOVL C00406 V=8.0
MOVL C00407 V=8.0
MOVL C00408 V=8.0
MOVL C00409 V=8.0
MOVL C00410 V=8.0
MOVL C00411 V=8.0
MOVL C00412 V=8.0
MOVL C00413 V=8.0
MOVL C00414 V=8.0
MOVL C00415 V=8.0
MOVL C00416 V=8.0
MOVL C00417 V=8.0
MOVL C00418 V=8.0
MOVL C00419 V=8.0
MOVL C00420 V=8.0
MOVL C00421 V=8.0
MOVL C00422 V=8.0
MOVL C00423 V=8.0
MOVL C00424 V=8.0
MOVL C00425 V=8.0
MOVL C00426 V=8.0
MOVL C00427 V=8.0
MOVL C00428 V=8.0
MOVL C00429 V=8.0
MOVL C00430 V=8.0
MOVL C00431 V=8.0
MOVL C00432 V=8.0
MOVL C00433 V=8.0
MOVL C00434 V=8.0
MOVL C00435 V=8.0
MOVL C00436 V=8.0
MOVL C00437 V=8.0
MOVL C00438 V=8.0
MOVL C00439 V=8.0
MOVL C00440 V=8.0
MOVJ C00441 VJ=0.78
MOVJ C00442 VJ=0.78
MOVJ C00443 VJ=0.78
MOVL C00444 V=8.0
MOVL C00445 V=8.0
MOVL C00446 V=8.0
MOVL C00447 V=8.0
MOVL C00448 V=8.0
MOVL C00449 V=8.0
MOVL C00450 V=8.0
MOVL C00451 V=8.0
MOVL C00452 V=8.0
MOVL C00453 V=8.0
MOVL C00454 V=8.0
MOVL C00455 V=8.0
MOVL C00456 V=8.0
MOVL C00457 V=8.0
MOVL C00458 V=8.0
MOVL C00459 V=8.0
MOVL C00460 V=8.0
MOVL C00461 V=8.0
MOVL C00462 V=8.0
MOVL C00463 V=8.0
MOVL C00464 V=8.0
MOVL C00465 V=8.0
MOVL C00466 V=8.0
MOVL C00467 V=8.0
MOVL C00468 V=8.0
MOVL C00469 V=8.0
MOVL C00470 V=8.0
MOVL C00471 V=8.0
MOVL C00472 V=8.0
MOVL C00473 V=8.0
MOVL C00474 V=8.0
MOVL C00475 V=8.0
MOVL C00476 V=8.0
MOVL C00477 V=8.0
MOVL C00478 V=8.0
MOVL C00479 V=8.0
MOVL C00480 V=8.0
MOVL C00481 V=8.0
MOVL C00482 V=8.0
MOVL C00483 V=8.0
MOVL C00484 V=8.0
MOVL C00485 V=8.0
MOVL C00486 V=8.0
MOVL C00487 V=8.0
MOVL C00488 V=8.0
MOVL C00489 V=8.0
MOVL C00490 V=8.0
MOVL C00491 V=8.0
MOVL C00492 V=8.0
MOVL C00493 V=8.0
MOVL C00494 V=8.0
MOVL C00495 V=8.0
MOVL C00496 V=8.0
MOVL C00497 V=8.0
MOVL C00498 V=8.0
MOVL C00499 V=8.0
MOVL C00500 V=8.0
MOVL C00501 V=8.0
MOVL C00502 V=8.0
MOVL C00503 V=8.0
MOVJ C00504 VJ=0.78
MOVJ C00505 VJ=0.78
MOVJ C00506 VJ=0.78
MOVL C00507 V=8.0
MOVL C00508 V=8.0
MOVL C00509 V=8.0
MOVL C00510 V=8.0
MOVL C00511 V=8.0
MOVL C00512 V=8.0
MOVL C00513 V=8.0
MOVL C00514 V=8.0
MOVL C00515 V=8.0
MOVL C00516 V=8.0
MOVL C00517 V=8.0
MOVL C00518 V=8.0
MOVL C00519 V=8.0
MOVL C00520 V=8.0
MOVL C00521 V=8.0
MOVL C00522 V=8.0
MOVL C00523 V=8.0
MOVL C00524 V=8.0
MOVL C00525 V=8.0
MOVL C00526 V=8.0
MOVL C00527 V=8.0
MOVL C00528 V=8.0
MOVL C00529 V=8.0
MOVL C00530 V=8.0
MOVL C00531 V=8.0
MOVL C00532 V=8.0
MOVL C00533 V=8.0
MOVL C00534 V=8.0
MOVL C00535 V=8.0
MOVL C00536 V=8.0
MOVL C00537 V=8.0
MOVL C00538 V=8.0
MOVL C00539 V=8.0
MOVL C00540 V=8.0
MOVL C00541 V=8.0
MOVL C00542 V=8.0
MOVL C00543 V=8.0
MOVL C00544 V=8.0
MOVL C00545 V=8.0
MOVL C00546 V=8.0
MOVL C00547 V=8.0
MOVL C00548 V=8.0
MOVL C00549 V=8.0
MOVL C00550 V=8.0
MOVL C00551 V=8.0
MOVL C00552 V=8.0
MOVL C00553 V=8.0
MOVL C00554 V=8.0
MOVL C00555 V=8.0
MOVL C00556 V=8.0
MOVL C00557 V=8.0
MOVL C00558 V=8.0
MOVL C00559 V=8.0
MOVL C00560 V=8.0
MOVL C00561 V=8.0
MOVL C00562 V=8.0
MOVL C00563 V=8.0
MOVL C00564 V=8.0
MOVL C00565 V=8.0
MOVL C00566 V=8.0
MOVJ C00567 VJ=0.78
MOVJ C00568 VJ=0.78
MOVJ C00569 VJ=0.78
MOVL C00570 V=8.0
MOVL C00571 V=8.0
MOVL C00572 V=8.0
MOVL C00573 V=8.0
MOVL C00574 V=8.0
MOVL C00575 V=8.0
MOVL C00576 V=8.0
MOVL C00577 V=8.0
MOVL C00578 V=8.0
MOVL C00579 V=8.0
MOVL C00580 V=8.0
MOVL C00581 V=8.0
MOVL C00582 V=8.0
MOVL C00583 V=8.0
MOVL C00584 V=8.0
MOVL C00585 V=8.0
MOVL C00586 V=8.0
MOVL C00587 V=8.0
MOVL C00588 V=8.0
MOVL C00589 V=8.0
MOVL C00590 V=8.0
MOVL C00591 V=8.0
MOVL C00592 V=8.0
MOVL C00593 V=8.0
MOVL C00594 V=8.0
MOVL C00595 V=8.0
MOVL C00596 V=8.0
MOVL C00597 V=8.0
MOVL C00598 V=8.0
MOVL C00599 V=8.0
MOVL C00600 V=8.0
MOVL C00601 V=8.0
MOVL C00602 V=8.0
MOVL C00603 V=8.0
MOVL C00604 V=8.0
MOVL C00605 V=8.0
MOVL C00606 V=8.0
MOVL C00607 V=8.0
MOVL C00608 V=8.0
MOVL C00609 V=8.0
MOVL C00610 V=8.0
MOVL C00611 V=8.0
MOVL C00612 V=8.0
MOVL C00613 V=8.0
MOVL C00614 V=8.0
MOVL C00615 V=8.0
MOVL C00616 V=8.0
MOVL C00617 V=8.0
MOVL C00618 V=8.0
MOVL C00619 V=8.0
MOVL C00620 V=8.0
MOVL C00621 V=8.0
MOVL C00622 V=8.0
MOVL C00623 V=8.0
MOVL C00624 V=8.0
MOVL C00625 V=8.0
MOVL C00626 V=8.0
MOVL C00627 V=8.0
MOVL C00628 V=8.0
MOVL C00629 V=8.0
MOVJ C00630 VJ=0.78
MOVJ C00631 VJ=0.78
MOVJ C00632 VJ=0.78
MOVL C00633 V=8.0
MOVL C00634 V=8.0
MOVL C00635 V=8.0
MOVL C00636 V=8.0
MOVL C00637 V=8.0
MOVL C00638 V=8.0
MOVL C00639 V=8.0
MOVL C00640 V=8.0
MOVL C00641 V=8.0
MOVL C00642 V=8.0
MOVL C00643 V=8.0
MOVL C00644 V=8.0
MOVL C00645 V=8.0
MOVL C00646 V=8.0
MOVL C00647 V=8.0
MOVL C00648 V=8.0
MOVL C00649 V=8.0
MOVL C00650 V=8.0
MOVL C00651 V=8.0
MOVL C00652 V=8.0
MOVL C00653 V=8.0
MOVL C00654 V=8.0
MOVL C00655 V=8.0
MOVL C00656 V=8.0
MOVL C00657 V=8.0
MOVL C00658 V=8.0
MOVL C00659 V=8.0
MOVL C00660 V=8.0
MOVL C00661 V=8.0
MOVL C00662 V=8.0
MOVL C00663 V=8.0
MOVL C00664 V=8.0
MOVL C00665 V=8.0
MOVL C00666 V=8.0
MOVL C00667 V=8.0
MOVL C00668 V=8.0
MOVL C00669 V=8.0
MOVL C00670 V=8.0
MOVL C00671 V=8.0
MOVL C00672 V=8.0
MOVL C00673 V=8.0
MOVL C00674 V=8.0
MOVL C00675 V=8.0
MOVL C00676 V=8.0
MOVL C00677 V=8.0
MOVL C00678 V=8.0
MOVL C00679 V=8.0
MOVL C00680 V=8.0
MOVL C00681 V=8.0
MOVL C00682 V=8.0
MOVL C00683 V=8.0
MOVL C00684 V=8.0
MOVL C00685 V=8.0
MOVL C00686 V=8.0
MOVL C00687 V=8.0
MOVL C00688 V=8.0
MOVL C00689 V=8.0
MOVL C00690 V=8.0
MOVL C00691 V=8.0
MOVL C00692 V=8.0
MOVJ C00693 VJ=0.78
MOVJ C00694 VJ=0.78
MOVJ C00695 VJ=0.78
MOVL C00696 V=8.0
MOVL C00697 V=8.0
MOVL C00698 V=8.0
MOVL C00699 V=8.0
MOVL C00700 V=8.0
MOVL C00701 V=8.0
MOVL C00702 V=8.0
MOVL C00703 V=8.0
MOVL C00704 V=8.0
MOVL C00705 V=8.0
MOVL C00706 V=8.0
MOVL C00707 V=8.0
MOVL C00708 V=8.0
MOVL C00709 V=8.0
MOVL C00710 V=8.0
MOVL C00711 V=8.0
MOVL C00712 V=8.0
MOVL C00713 V=8.0
MOVL C00714 V=8.0
MOVL C00715 V=8.0
MOVL C00716 V=8.0
MOVL C00717 V=8.0
MOVL C00718 V=8.0
MOVL C00719 V=8.0
MOVL C00720 V=8.0
MOVL C00721 V=8.0
MOVL C00722 V=8.0
MOVL C00723 V=8.0
MOVL C00724 V=8.0
MOVL C00725 V=8.0
MOVL C00726 V=8.0
MOVL C00727 V=8.0
MOVL C00728 V=8.0
MOVL C00729 V=8.0
MOVL C00730 V=8.0
MOVL C00731 V=8.0
MOVL C00732 V=8.0
MOVL C00733 V=8.0
MOVL C00734 V=8.0
MOVL C00735 V=8.0
MOVL C00736 V=8.0
MOVL C00737 V=8.0
MOVL C00738 V=8.0
MOVL C00739 V=8.0
MOVL C00740 V=8.0
MOVL C00741 V=8.0
MOVL C00742 V=8.0
MOVL C00743 V=8.0
MOVL C00744 V=8.0
MOVL C00745 V=8.0
MOVL C00746 V=8.0
MOVL C00747 V=8.0
MOVL C00748 V=8.0
MOVL C00749 V=8.0
MOVL C00750 V=8.0
MOVL C00751 V=8.0
MOVL C00752 V=8.0
MOVL C00753 V=8.0
MOVL C00754 V=8.0
MOVL C00755 V=8.0
MOVJ C00756 VJ=0.78
MOVJ C00757 VJ=0.78
MOVJ C00758 VJ=0.78
MOVL C00759 V=8.0
MOVL C00760 V=8.0
MOVL C00761 V=8.0
MOVL C00762 V=8.0
MOVL C00763 V=8.0
MOVL C00764 V=8.0
MOVL C00765 V=8.0
MOVL C00766 V=8.0
MOVL C00767 V=8.0
MOVL C00768 V=8.0
MOVL C00769 V=8.0
MOVL C00770 V=8.0
MOVL C00771 V=8.0
MOVL C00772 V=8.0
MOVL C00773 V=8.0
MOVL C00774 V=8.0
MOVL C00775 V=8.0
MOVL C00776 V=8.0
MOVL C00777 V=8.0
MOVL C00778 V=8.0
MOVL C00779 V=8.0
MOVL C00780 V=8.0
MOVL C00781 V=8.0
MOVL C00782 V=8.0
MOVL C00783 V=8.0
MOVL C00784 V=8.0
MOVL C00785 V=8.0
MOVL C00786 V=8.0
MOVL C00787 V=8.0
MOVL C00788 V=8.0
MOVL C00789 V=8.0
MOVL C00790 V=8.0
MOVL C00791 V=8.0
MOVL C00792 V=8.0
MOVL C00793 V=8.0
MOVL C00794 V=8.0
MOVL C00795 V=8.0
MOVL C00796 V=8.0
MOVL C00797 V=8.0
MOVL C00798 V=8.0
MOVL C00799 V=8.0
MOVL C00800 V=8.0
MOVL C00801 V=8.0
MOVL C00802 V=8.0
MOVL C00803 V=8.0
MOVL C00804 V=8.0
MOVL C00805 V=8.0
MOVL C00806 V=8.0
MOVL C00807 V=8.0
MOVL C00808 V=8.0
MOVL C00809 V=8.0
MOVL C00810 V=8.0
MOVL C00811 V=8.0
MOVL C00812 V=8.0
MOVL C00813 V=8.0
MOVL C00814 V=8.0
MOVL C00815 V=8.0
MOVL C00816 V=8.0
MOVL C00817 V=8.0
MOVL C00818 V=8.0
MOVJ C00819 VJ=0.78
MOVJ C00820 VJ=0.78
MOVJ C00821 VJ=0.78
MOVL C00822 V=8.0
MOVL C00823 V=8.0
MOVL C00824 V=8.0
MOVL C00825 V=8.0
MOVL C00826 V=8.0
MOVL C00827 V=8.0
MOVL C00828 V=8.0
MOVL C00829 V=8.0
MOVL C00830 V=8.0
MOVL C00831 V=8.0
MOVL C00832 V=8.0
MOVL C00833 V=8.0
MOVL C00834 V=8.0
MOVL C00835 V=8.0
MOVL C00836 V=8.0
MOVL C00837 V=8.0
MOVL C00838 V=8.0
MOVL C00839 V=8.0
MOVL C00840 V=8.0
MOVL C00841 V=8.0
MOVL C00842 V=8.0
MOVL C00843 V=8.0
MOVL C00844 V=8.0
MOVL C00845 V=8.0
MOVL C00846 V=8.0
MOVL C00847 V=8.0
MOVL C00848 V=8.0
MOVL C00849 V=8.0
MOVL C00850 V=8.0
MOVL C00851 V=8.0
MOVL C00852 V=8.0
MOVL C00853 V=8.0
MOVL C00854 V=8.0
MOVL C00855 V=8.0
MOVL C00856 V=8.0
MOVL C00857 V=8.0
MOVL C00858 V=8.0
MOVL C00859 V=8.0
MOVL C00860 V=8.0
MOVL C00861 V=8.0
MOVL C00862 V=8.0
MOVL C00863 V=8.0
MOVL C00864 V=8.0
MOVL C00865 V=8.0
MOVL C00866 V=8.0
MOVL C00867 V=8.0
MOVL C00868 V=8.0
MOVL C00869 V=8.0
MOVL C00870 V=8.0
MOVL C00871 V=8.0
MOVL C00872 V=8.0
MOVL C00873 V=8.0
MOVL C00874 V=8.0
MOVL C00875 V=8.0
MOVL C00876 V=8.0
MOVL C00877 V=8.0
MOVL C00878 V=8.0
MOVL C00879 V=8.0
MOVL C00880 V=8.0
MOVL C00881 V=8.0
MOVJ C00882 VJ=0.78
MOVJ C00883 VJ=0.78
MOVJ C00884 VJ=0.78
MOVL C00885 V=8.0
MOVL C00886 V=8.0
MOVL C00887 V=8.0
MOVL C00888 V=8.0
MOVL C00889 V=8.0
MOVL C00890 V=8.0
MOVL C00891 V=8.0
MOVL C00892 V=8.0
MOVL C00893 V=8.0
MOVL C00894 V=8.0
MOVL C00895 V=8.0
MOVL C00896 V=8.0
MOVL C00897 V=8.0
MOVL C00898 V=8.0
MOVL C00899 V=8.0
MOVL C00900 V=8.0
MOVL C00901 V=8.0
MOVL C00902 V=8.0
MOVL C00903 V=8.0
MOVL C00904 V=8.0
MOVL C00905 V=8.0
MOVL C00906 V=8.0
MOVL C00907 V=8.0
MOVL C00908 V=8.0
MOVL C00909 V=8.0
MOVL C00910 V=8.0
MOVL C00911 V=8.0
MOVL C00912 V=8.0
MOVL C00913 V=8.0
MOVL C00914 V=8.0
MOVL C00915 V=8.0
MOVL C00916 V=8.0
MOVL C00917 V=8.0
MOVL C00918 V=8.0
MOVL C00919 V=8.0
MOVL C00920 V=8.0
MOVL C00921 V=8.0
MOVL C00922 V=8.0
MOVL C00923 V=8.0
MOVL C00924 V=8.0
MOVL C00925 V=8.0
MOVL C00926 V=8.0
MOVL C00927 V=8.0
MOVL C00928 V=8.0
MOVL C00929 V=8.0
MOVL C00930 V=8.0
MOVL C00931 V=8.0
MOVL C00932 V=8.0
MOVL C00933 V=8.0
MOVL C00934 V=8.0
MOVL C00935 V=8.0
MOVL C00936 V=8.0
MOVL C00937 V=8.0
MOVL C00938 V=8.0
MOVL C00939 V=8.0
MOVL C00940 V=8.0
MOVL C00941 V=8.0
MOVL C00942 V=8.0
MOVL C00943 V=8.0
MOVL C00944 V=8.0
MOVJ C00945 VJ=0.78
MOVJ C00946 VJ=0.78
MOVJ C00947 VJ=0.78
MOVL C00948 V=8.0
MOVL C00949 V=8.0
MOVL C00950 V=8.0
MOVL C00951 V=8.0
MOVL C00952 V=8.0
MOVL C00953 V=8.0
MOVL C00954 V=8.0
MOVL C00955 V=8.0
MOVL C00956 V=8.0
MOVL C00957 V=8.0
MOVL C00958 V=8.0
MOVL C00959 V=8.0
MOVL C00960 V=8.0
MOVL C00961 V=8.0
MOVL C00962 V=8.0
MOVL C00963 V=8.0
MOVL C00964 V=8.0
MOVL C00965 V=8.0
MOVL C00966 V=8.0
MOVL C00967 V=8.0
MOVL C00968 V=8.0
MOVL C00969 V=8.0
MOVL C00970 V=8.0
MOVL C00971 V=8.0
MOVL C00972 V=8.0
MOVL C00973 V=8.0
MOVL C00974 V=8.0
MOVL C00975 V=8.0
MOVL C00976 V=8.0
MOVL C00977 V=8.0
MOVL C00978 V=8.0
MOVL C00979 V=8.0
MOVL C00980 V=8.0
MOVL C00981 V=8.0
MOVL C00982 V=8.0
MOVL C00983 V=8.0
MOVL C00984 V=8.0
MOVL C00985 V=8.0
MOVL C00986 V=8.0
MOVL C00987 V=8.0
MOVL C00988 V=8.0
MOVL C00989 V=8.0
MOVL C00990 V=8.0
MOVL C00991 V=8.0
MOVL C00992 V=8.0
MOVL C00993 V=8.0
MOVL C00994 V=8.0
MOVL C00995 V=8.0
MOVL C00996 V=8.0
MOVL C00997 V=8.0
MOVL C00998 V=8.0
MOVL C00999 V=8.0
MOVL C01000 V=8.0
MOVL C01001 V=8.0
MOVL C01002 V=8.0
MOVL C01003 V=8.0
MOVL C01004 V=8.0
MOVL C01005 V=8.0
MOVL C01006 V=8.0
MOVL C01007 V=8.0
MOVJ C01008 VJ=0.78
MOVJ C01009 VJ=0.78
MOVJ C01010 VJ=0.78
MOVL C01011 V=8.0
MOVL C01012 V=8.0
MOVL C01013 V=8.0
MOVL C01014 V=8.0
MOVL C01015 V=8.0
MOVL C01016 V=8.0
MOVL C01017 V=8.0
MOVL C01018 V=8.0
MOVL C01019 V=8.0
MOVL C01020 V=8.0
MOVL C01021 V=8.0
MOVL C01022 V=8.0
MOVL C01023 V=8.0
MOVL C01024 V=8.0
MOVL C01025 V=8.0
MOVL C01026 V=8.0
MOVL C01027 V=8.0
MOVL C01028 V=8.0
MOVL C01029 V=8.0
MOVL C01030 V=8.0
MOVL C01031 V=8.0
MOVL C01032 V=8.0
MOVL C01033 V=8.0
MOVL C01034 V=8.0
MOVL C01035 V=8.0
MOVL C01036 V=8.0
MOVL C01037 V=8.0
MOVL C01038 V=8.0
MOVL C01039 V=8.0
MOVL C01040 V=8.0
MOVL C01041 V=8.0
MOVL C01042 V=8.0
MOVL C01043 V=8.0
MOVL C01044 V=8.0
MOVL C01045 V=8.0
MOVL C01046 V=8.0
MOVL C01047 V=8.0
MOVL C01048 V=8.0
MOVL C01049 V=8.0
MOVL C01050 V=8.0
MOVL C01051 V=8.0
MOVL C01052 V=8.0
MOVL C01053 V=8.0
MOVL C01054 V=8.0
MOVL C01055 V=8.0
MOVL C01056 V=8.0
MOVL C01057 V=8.0
MOVL C01058 V=8.0
MOVL C01059 V=8.0
MOVL C01060 V=8.0
MOVL C01061 V=8.0
MOVL C01062 V=8.0
MOVL C01063 V=8.0
MOVL C01064 V=8.0
MOVL C01065 V=8.0
MOVL C01066 V=8.0
MOVL C01067 V=8.0
MOVL C01068 V=8.0
MOVL C01069 V=8.0
MOVL C01070 V=8.0
MOVJ C01071 VJ=0.78
MOVJ C01072 VJ=0.78
MOVJ C01073 VJ=0.78
MOVL C01074 V=8.0
MOVL C01075 V=8.0
MOVL C01076 V=8.0
MOVL C01077 V=8.0
MOVL C01078 V=8.0
MOVL C01079 V=8.0
MOVL C01080 V=8.0
MOVL C01081 V=8.0
MOVL C01082 V=8.0
MOVL C01083 V=8.0
MOVL C01084 V=8.0
MOVL C01085 V=8.0
MOVL C01086 V=8.0
MOVL C01087 V=8.0
MOVL C01088 V=8.0
MOVL C01089 V=8.0
MOVL C01090 V=8.0
MOVL C01091 V=8.0
MOVL C01092 V=8.0
MOVL C01093 V=8.0
MOVL C01094 V=8.0
MOVL C01095 V=8.0
MOVL C01096 V=8.0
MOVL C01097 V=8.0
MOVL C01098 V=8.0
MOVL C01099 V=8.0
MOVL C01100 V=8.0
MOVL C01101 V=8.0
MOVL C01102 V=8.0
MOVL C01103 V=8.0
MOVL C01104 V=8.0
MOVL C01105 V=8.0
MOVL C01106 V=8.0
MOVL C01107 V=8.0
MOVL C01108 V=8.0
MOVL C01109 V=8.0
MOVL C01110 V=8.0
MOVL C01111 V=8.0
MOVL C01112 V=8.0
MOVL C01113 V=8.0
MOVL C01114 V=8.0
MOVL C01115 V=8.0
MOVL C01116 V=8.0
MOVL C01117 V=8.0
MOVL C01118 V=8.0
MOVL C01119 V=8.0
MOVL C01120 V=8.0
MOVL C01121 V=8.0
MOVL C01122 V=8.0
MOVL C01123 V=8.0
MOVL C01124 V=8.0
MOVL C01125 V=8.0
MOVL C01126 V=8.0
MOVL C01127 V=8.0
MOVL C01128 V=8.0
MOVL C01129 V=8.0
MOVL C01130 V=8.0
MOVL C01131 V=8.0
MOVL C01132 V=8.0
MOVL C01133 V=8.0
MOVJ C01134 VJ=0.78
MOVJ C01135 VJ=0.78
MOVJ C01136 VJ=0.78
MOVL C01137 V=8.0
MOVL C01138 V=8.0
MOVL C01139 V=8.0
MOVL C01140 V=8.0
MOVL C01141 V=8.0
MOVL C01142 V=8.0
MOVL C01143 V=8.0
MOVL C01144 V=8.0
MOVL C01145 V=8.0
MOVL C01146 V=8.0
MOVL C01147 V=8.0
MOVL C01148 V=8.0
MOVL C01149 V=8.0
MOVL C01150 V=8.0
MOVL C01151 V=8.0
MOVL C01152 V=8.0
MOVL C01153 V=8.0
MOVL C01154 V=8.0
MOVL C01155 V=8.0
MOVL C01156 V=8.0
MOVL C01157 V=8.0
MOVL C01158 V=8.0
MOVL C01159 V=8.0
MOVL C01160 V=8.0
MOVL C01161 V=8.0
MOVL C01162 V=8.0
MOVL C01163 V=8.0
MOVL C01164 V=8.0
MOVL C01165 V=8.0
MOVL C01166 V=8.0
MOVL C01167 V=8.0
MOVL C01168 V=8.0
MOVL C01169 V=8.0
MOVL C01170 V=8.0
MOVL C01171 V=8.0
MOVL C01172 V=8.0
MOVL C01173 V=8.0
MOVL C01174 V=8.0
MOVL C01175 V=8.0
MOVL C01176 V=8.0
MOVL C01177 V=8.0
MOVL C01178 V=8.0
MOVL C01179 V=8.0
MOVL C01180 V=8.0
MOVL C01181 V=8.0
MOVL C01182 V=8.0
MOVL C01183 V=8.0
MOVL C01184 V=8.0
MOVL C01185 V=8.0
MOVL C01186 V=8.0
MOVL C01187 V=8.0
MOVL C01188 V=8.0
MOVL C01189 V=8.0
MOVL C01190 V=8.0
MOVL C01191 V=8.0
MOVL C01192 V=8.0
MOVL C01193 V=8.0
MOVL C01194 V=8.0
MOVL C01195 V=8.0
MOVL C01196 V=8.0
MOVJ C01197 VJ=0.78
MOVJ C01198 VJ=0.78
MOVJ C01199 VJ=0.78
MOVL C01200 V=8.0
MOVL C01201 V=8.0
MOVL C01202 V=8.0
MOVL C01203 V=8.0
MOVL C01204 V=8.0
MOVL C01205 V=8.0
MOVL C01206 V=8.0
MOVL C01207 V=8.0
MOVL C01208 V=8.0
MOVL C01209 V=8.0
MOVL C01210 V=8.0
MOVL C01211 V=8.0
MOVL C01212 V=8.0
MOVL C01213 V=8.0
MOVL C01214 V=8.0
MOVL C01215 V=8.0
MOVL C01216 V=8.0
MOVL C01217 V=8.0
MOVL C01218 V=8.0
MOVL C01219 V=8.0
MOVL C01220 V=8.0
MOVL C01221 V=8.0
MOVL C01222 V=8.0
MOVL C01223 V=8.0
MOVL C01224 V=8.0
MOVL C01225 V=8.0
MOVL C01226 V=8.0
MOVL C01227 V=8.0
MOVL C01228 V=8.0
MOVL C01229 V=8.0
MOVL C01230 V=8.0
MOVL C01231 V=8.0
MOVL C01232 V=8.0
MOVL C01233 V=8.0
MOVL C01234 V=8.0
MOVL C01235 V=8.0
MOVL C01236 V=8.0
MOVL C01237 V=8.0
MOVL C01238 V=8.0
MOVL C01239 V=8.0
MOVL C01240 V=8.0
MOVL C01241 V=8.0
MOVL C01242 V=8.0
MOVL C01243 V=8.0
MOVL C01244 V=8.0
MOVL C01245 V=8.0
MOVL C01246 V=8.0
MOVL C01247 V=8.0
MOVL C01248 V=8.0
MOVL C01249 V=8.0
MOVL C01250 V=8.0
MOVL C01251 V=8.0
MOVL C01252 V=8.0
MOVL C01253 V=8.0
MOVL C01254 V=8.0
MOVL C01255 V=8.0
MOVL C01256 V=8.0
MOVL C01257 V=8.0
MOVL C01258 V=8.0
MOVL C01259 V=8.0
MOVJ C01260 VJ=0.78
MOVJ C01261 VJ=0.78
MOVJ C01262 VJ=0.78
MOVL C01263 V=8.0
MOVL C01264 V=8.0
MOVL C01265 V=8.0
MOVL C01266 V=8.0
MOVL C01267 V=8.0
MOVL C01268 V=8.0
MOVL C01269 V=8.0
MOVL C01270 V=8.0
MOVL C01271 V=8.0
MOVL C01272 V=8.0
MOVL C01273 V=8.0
MOVL C01274 V=8.0
MOVL C01275 V=8.0
MOVL C01276 V=8.0
MOVL C01277 V=8.0
MOVL C01278 V=8.0
MOVL C01279 V=8.0
MOVL C01280 V=8.0
MOVL C01281 V=8.0
MOVL C01282 V=8.0
MOVL C01283 V=8.0
MOVL C01284 V=8.0
MOVL C01285 V=8.0
MOVL C01286 V=8.0
MOVL C01287 V=8.0
MOVL C01288 V=8.0
MOVL C01289 V=8.0
MOVL C01290 V=8.0
MOVL C01291 V=8.0
MOVL C01292 V=8.0
MOVL C01293 V=8.0
MOVL C01294 V=8.0
MOVL C01295 V=8.0
MOVL C01296 V=8.0
MOVL C01297 V=8.0
MOVL C01298 V=8.0
MOVL C01299 V=8.0
MOVL C01300 V=8.0
MOVL C01301 V=8.0
MOVL C01302 V=8.0
MOVL C01303 V=8.0
MOVL C01304 V=8.0
MOVL C01305 V=8.0
MOVL C01306 V=8.0
MOVL C01307 V=8.0
MOVL C01308 V=8.0
MOVL C01309 V=8.0
MOVL C01310 V=8.0
MOVL C01311 V=8.0
MOVL C01312 V=8.0
MOVL C01313 V=8.0
MOVL C01314 V=8.0
MOVL C01315 V=8.0
MOVL C01316 V=8.0
MOVL C01317 V=8.0
MOVL C01318 V=8.0
MOVL C01319 V=8.0
MOVL C01320 V=8.0
MOVL C01321 V=8.0
MOVL C01322 V=8.0
MOVJ C01323 VJ=0.78
MOVJ C01324 VJ=0.78
MOVJ C01325 VJ=0.78
MOVL C01326 V=8.0
MOVL C01327 V=8.0
MOVL C01328 V=8.0
MOVL C01329 V=8.0
MOVL C01330 V=8.0
MOVL C01331 V=8.0
MOVL C01332 V=8.0
MOVL C01333 V=8.0
MOVL C01334 V=8.0
MOVL C01335 V=8.0
MOVL C01336 V=8.0
MOVL C01337 V=8.0
MOVL C01338 V=8.0
MOVL C01339 V=8.0
MOVL C01340 V=8.0
MOVL C01341 V=8.0
MOVL C01342 V=8.0
MOVL C01343 V=8.0
MOVL C01344 V=8.0
MOVL C01345 V=8.0
MOVL C01346 V=8.0
MOVL C01347 V=8.0
MOVL C01348 V=8.0
MOVL C01349 V=8.0
MOVL C01350 V=8.0
MOVL C01351 V=8.0
MOVL C01352 V=8.0
MOVL C01353 V=8.0
MOVL C01354 V=8.0
MOVL C01355 V=8.0
MOVL C01356 V=8.0
MOVL C01357 V=8.0
MOVL C01358 V=8.0
MOVL C01359 V=8.0
MOVL C01360 V=8.0
MOVL C01361 V=8.0
MOVL C01362 V=8.0
MOVL C01363 V=8.0
MOVL C01364 V=8.0
MOVL C01365 V=8.0
MOVL C01366 V=8.0
MOVL C01367 V=8.0
MOVL C01368 V=8.0
MOVL C01369 V=8.0
MOVL C01370 V=8.0
MOVL C01371 V=8.0
MOVL C01372 V=8.0
MOVL C01373 V=8.0
MOVL C01374 V=8.0
MOVL C01375 V=8.0
MOVL C01376 V=8.0
MOVL C01377 V=8.0
MOVL C01378 V=8.0
MOVL C01379 V=8.0
MOVL C01380 V=8.0
MOVL C01381 V=8.0
MOVL C01382 V=8.0
MOVL C01383 V=8.0
MOVL C01384 V=8.0
MOVL C01385 V=8.0
MOVJ C01386 VJ=0.78
MOVJ C01387 VJ=0.78
MOVJ C01388 VJ=0.78
MOVL C01389 V=8.0
MOVL C01390 V=8.0
MOVL C01391 V=8.0
MOVL C01392 V=8.0
MOVL C01393 V=8.0
MOVL C01394 V=8.0
MOVL C01395 V=8.0
MOVL C01396 V=8.0
MOVL C01397 V=8.0
MOVL C01398 V=8.0
MOVL C01399 V=8.0
MOVL C01400 V=8.0
MOVL C01401 V=8.0
MOVL C01402 V=8.0
MOVL C01403 V=8.0
MOVL C01404 V=8.0
MOVL C01405 V=8.0
MOVL C01406 V=8.0
MOVL C01407 V=8.0
MOVL C01408 V=8.0
MOVL C01409 V=8.0
MOVL C01410 V=8.0
MOVL C01411 V=8.0
MOVL C01412 V=8.0
MOVL C01413 V=8.0
MOVL C01414 V=8.0
MOVL C01415 V=8.0
MOVL C01416 V=8.0
MOVL C01417 V=8.0
MOVL C01418 V=8.0
MOVL C01419 V=8.0
MOVL C01420 V=8.0
MOVL C01421 V=8.0
MOVL C01422 V=8.0
MOVL C01423 V=8.0
MOVL C01424 V=8.0
MOVL C01425 V=8.0
MOVL C01426 V=8.0
MOVL C01427 V=8.0
MOVL C01428 V=8.0
MOVL C01429 V=8.0
MOVL C01430 V=8.0
MOVL C01431 V=8.0
MOVL C01432 V=8.0
MOVL C01433 V=8.0
MOVL C01434 V=8.0
MOVL C01435 V=8.0
MOVL C01436 V=8.0
MOVL C01437 V=8.0
MOVL C01438 V=8.0
MOVL C01439 V=8.0
MOVL C01440 V=8.0
MOVL C01441 V=8.0
MOVL C01442 V=8.0
MOVL C01443 V=8.0
MOVL C01444 V=8.0
MOVL C01445 V=8.0
MOVL C01446 V=8.0
MOVL C01447 V=8.0
MOVL C01448 V=8.0
MOVJ C01449 VJ=0.78
MOVJ C01450 VJ=0.78
MOVJ C01451 VJ=0.78
MOVL C01452 V=8.0
MOVL C01453 V=8.0
MOVL C01454 V=8.0
MOVL C01455 V=8.0
MOVL C01456 V=8.0
MOVL C01457 V=8.0
MOVL C01458 V=8.0
MOVL C01459 V=8.0
MOVL C01460 V=8.0
MOVL C01461 V=8.0
MOVL C01462 V=8.0
MOVL C01463 V=8.0
MOVL C01464 V=8.0
MOVL C01465 V=8.0
MOVL C01466 V=8.0
MOVL C01467 V=8.0
MOVL C01468 V=8.0
MOVL C01469 V=8.0
MOVL C01470 V=8.0
MOVL C01471 V=8.0
MOVL C01472 V=8.0
MOVL C01473 V=8.0
MOVL C01474 V=8.0
MOVL C01475 V=8.0
MOVL C01476 V=8.0
MOVL C01477 V=8.0
MOVL C01478 V=8.0
MOVL C01479 V=8.0
MOVL C01480 V=8.0
MOVL C01481 V=8.0
MOVL C01482 V=8.0
MOVL C01483 V=8.0
MOVL C01484 V=8.0
MOVL C01485 V=8.0
MOVL C01486 V=8.0
MOVL C01487 V=8.0
MOVL C01488 V=8.0
MOVL C01489 V=8.0
MOVL C01490 V=8.0
MOVL C01491 V=8.0
MOVL C01492 V=8.0
MOVL C01493 V=8.0
MOVL C01494 V=8.0
MOVL C01495 V=8.0
MOVL C01496 V=8.0
MOVL C01497 V=8.0
MOVL C01498 V=8.0
MOVL C01499 V=8.0
MOVL C01500 V=8.0
MOVL C01501 V=8.0
MOVL C01502 V=8.0
MOVL C01503 V=8.0
MOVL C01504 V=8.0
MOVL C01505 V=8.0
MOVL C01506 V=8.0
MOVL C01507 V=8.0
MOVL C01508 V=8.0
MOVL C01509 V=8.0
MOVL C01510 V=8.0
MOVL C01511 V=8.0
MOVJ C01512 VJ=0.78
MOVJ C01513 VJ=0.78
MOVJ C01514 VJ=0.78
MOVL C01515 V=8.0
MOVL C01516 V=8.0
MOVL C01517 V=8.0
MOVL C01518 V=8.0
MOVL C01519 V=8.0
MOVL C01520 V=8.0
MOVL C01521 V=8.0
MOVL C01522 V=8.0
MOVL C01523 V=8.0
MOVL C01524 V=8.0
MOVL C01525 V=8.0
MOVL C01526 V=8.0
MOVL C01527 V=8.0
MOVL C01528 V=8.0
MOVL C01529 V=8.0
MOVL C01530 V=8.0
MOVL C01531 V=8.0
MOVL C01532 V=8.0
MOVL C01533 V=8.0
MOVL C01534 V=8.0
MOVL C01535 V=8.0
MOVL C01536 V=8.0
MOVL C01537 V=8.0
MOVL C01538 V=8.0
MOVL C01539 V=8.0
MOVL C01540 V=8.0
MOVL C01541 V=8.0
MOVL C01542 V=8.0
MOVL C01543 V=8.0
MOVL C01544 V=8.0
MOVL C01545 V=8.0
MOVL C01546 V=8.0
MOVL C01547 V=8.0
MOVL C01548 V=8.0
MOVL C01549 V=8.0
MOVL C01550 V=8.0
MOVL C01551 V=8.0
MOVL C01552 V=8.0
MOVL C01553 V=8.0
MOVL C01554 V=8.0
MOVL C01555 V=8.0
MOVL C01556 V=8.0
MOVL C01557 V=8.0
MOVL C01558 V=8.0
MOVL C01559 V=8.0
MOVL C01560 V=8.0
MOVL C01561 V=8.0
MOVL C01562 V=8.0
MOVL C01563 V=8.0
MOVL C01564 V=8.0
MOVL C01565 V=8.0
MOVL C01566 V=8.0
MOVL C01567 V=8.0
MOVL C01568 V=8.0
MOVL C01569 V=8.0
MOVL C01570 V=8.0
MOVL C01571 V=8.0
MOVL C01572 V=8.0
MOVL C01573 V=8.0
MOVL C01574 V=8.0
MOVJ C01575 VJ=0.78
END
